# B&R Automation Studio project A2019059_Linka_Power_CP (part 38)

#### TesterKomunikacia.st
```iecst
ACTION TesterKomunikacia:

	//Vstupy z Testera do PLC//
	AteqLeakageTester_A.Stav_RESET_DONE:= AteqLeakageTester_A.Profinet_PLC_INPUTS[1].0;
	AteqLeakageTester_A.Stav_START_DONE:= AteqLeakageTester_A.Profinet_PLC_INPUTS[1].1;
	AteqLeakageTester_A.Stav_ZmenaProgramu_DONE:= AteqLeakageTester_A.Profinet_PLC_INPUTS[1].3;
	AteqLeakageTester_A.Stav_CitanieParametrov_OK:= AteqLeakageTester_A.Profinet_PLC_INPUTS[1].5;

    AteqLeakageTester_A.Stav_CitanieParametrov_ERROR:= AteqLeakageTester_A.Profinet_PLC_INPUTS[3].5;

	AteqLeakageTester_A.CisloAktualnehoProgramu.0:= AteqLeakageTester_A.Profinet_PLC_INPUTS[7].0;
	AteqLeakageTester_A.CisloAktualnehoProgramu.1:= AteqLeakageTester_A.Profinet_PLC_INPUTS[7].1;
	AteqLeakageTester_A.CisloAktualnehoProgramu.2:= AteqLeakageTester_A.Profinet_PLC_INPUTS[7].2;
	AteqLeakageTester_A.CisloAktualnehoProgramu.3:= AteqLeakageTester_A.Profinet_PLC_INPUTS[7].3;
	AteqLeakageTester_A.CisloAktualnehoProgramu.4:= AteqLeakageTester_A.Profinet_PLC_INPUTS[7].4;
	AteqLeakageTester_A.CisloAktualnehoProgramu.5:= AteqLeakageTester_A.Profinet_PLC_INPUTS[7].5;
	AteqLeakageTester_A.CisloAktualnehoProgramu.6:= AteqLeakageTester_A.Profinet_PLC_INPUTS[7].6;
	AteqLeakageTester_A.CisloAktualnehoProgramu.7:= AteqLeakageTester_A.Profinet_PLC_INPUTS[7].7;

	AteqLeakageTester_A.CisloAktualnehoProgramu.8:= AteqLeakageTester_A.Profinet_PLC_INPUTS[8].0;
	AteqLeakageTester_A.CisloAktualnehoProgramu.9:= AteqLeakageTester_A.Profinet_PLC_INPUTS[8].1;
	AteqLeakageTester_A.CisloAktualnehoProgramu.10:= AteqLeakageTester_A.Profinet_PLC_INPUTS[8].2;
	AteqLeakageTester_A.CisloAktualnehoProgramu.11:= AteqLeakageTester_A.Profinet_PLC_INPUTS[8].3;
	AteqLeakageTester_A.CisloAktualnehoProgramu.12:= AteqLeakageTester_A.Profinet_PLC_INPUTS[8].4;
	AteqLeakageTester_A.CisloAktualnehoProgramu.13:= AteqLeakageTester_A.Profinet_PLC_INPUTS[8].5;
	AteqLeakageTester_A.CisloAktualnehoProgramu.14:= AteqLeakageTester_A.Profinet_PLC_INPUTS[8].6;
	AteqLeakageTester_A.CisloAktualnehoProgramu.15:= AteqLeakageTester_A.Profinet_PLC_INPUTS[8].7;

	AteqLeakageTester_A.VysledokTestovania_OK:= AteqLeakageTester_A.Profinet_PLC_INPUTS[13].0;
	AteqLeakageTester_A.VysledokTestovania_NG:= AteqLeakageTester_A.Profinet_PLC_INPUTS[13].1;
	AteqLeakageTester_A.Stav_ERROR:= AteqLeakageTester_A.Profinet_PLC_INPUTS[13].3;
	AteqLeakageTester_A.Stav_READY:= AteqLeakageTester_A.Profinet_PLC_INPUTS[13].5;

    AteqLeakageTester_A.ReadParameter_1.0:= AteqLeakageTester_A.Profinet_PLC_INPUTS[35].0;
    AteqLeakageTester_A.ReadParameter_1.1:= AteqLeakageTester_A.Profinet_PLC_INPUTS[35].1;
    AteqLeakageTester_A.ReadParameter_1.2:= AteqLeakageTester_A.Profinet_PLC_INPUTS[35].2;
    AteqLeakageTester_A.ReadParameter_1.3:= AteqLeakageTester_A.Profinet_PLC_INPUTS[35].3;
    AteqLeakageTester_A.ReadParameter_1.4:= AteqLeakageTester_A.Profinet_PLC_INPUTS[35].4;
    AteqLeakageTester_A.ReadParameter_1.5:= AteqLeakageTester_A.Profinet_PLC_INPUTS[35].5;
    AteqLeakageTester_A.ReadParameter_1.6:= AteqLeakageTester_A.Profinet_PLC_INPUTS[35].6;
    AteqLeakageTester_A.ReadParameter_1.7:= AteqLeakageTester_A.Profinet_PLC_INPUTS[35].7;
    AteqLeakageTester_A.ReadParameter_1.8:= AteqLeakageTester_A.Profinet_PLC_INPUTS[36].0;
    AteqLeakageTester_A.ReadParameter_1.9:= AteqLeakageTester_A.Profinet_PLC_INPUTS[36].1;
    AteqLeakageTester_A.ReadParameter_1.10:= AteqLeakageTester_A.Profinet_PLC_INPUTS[36].2;
    AteqLeakageTester_A.ReadParameter_1.11:= AteqLeakageTester_A.Profinet_PLC_INPUTS[36].3;
    AteqLeakageTester_A.ReadParameter_1.12:= AteqLeakageTester_A.Profinet_PLC_INPUTS[36].4;
    AteqLeakageTester_A.ReadParameter_1.13:= AteqLeakageTester_A.Profinet_PLC_INPUTS[36].5;
    AteqLeakageTester_A.ReadParameter_1.14:= AteqLeakageTester_A.Profinet_PLC_INPUTS[36].6;
    AteqLeakageTester_A.ReadParameter_1.15:= AteqLeakageTester_A.Profinet_PLC_INPUTS[36].7;

    AteqLeakageTester_A.ReadParameter_2.0:= AteqLeakageTester_A.Profinet_PLC_INPUTS[41].0;
    AteqLeakageTester_A.ReadParameter_2.1:= AteqLeakageTester_A.Profinet_PLC_INPUTS[41].1;
    AteqLeakageTester_A.ReadParameter_2.2:= AteqLeakageTester_A.Profinet_PLC_INPUTS[41].2;
    AteqLeakageTester_A.ReadParameter_2.3:= AteqLeakageTester_A.Profinet_PLC_INPUTS[41].3;
    AteqLeakageTester_A.ReadParameter_2.4:= AteqLeakageTester_A.Profinet_PLC_INPUTS[41].4;
    AteqLeakageTester_A.ReadParameter_2.5:= AteqLeakageTester_A.Profinet_PLC_INPUTS[41].5;
    AteqLeakageTester_A.ReadParameter_2.6:= AteqLeakageTester_A.Profinet_PLC_INPUTS[41].6;
    AteqLeakageTester_A.ReadParameter_2.7:= AteqLeakageTester_A.Profinet_PLC_INPUTS[41].7;
    AteqLeakageTester_A.ReadParameter_2.8:= AteqLeakageTester_A.Profinet_PLC_INPUTS[42].0;
    AteqLeakageTester_A.ReadParameter_2.9:= AteqLeakageTester_A.Profinet_PLC_INPUTS[42].1;
    AteqLeakageTester_A.ReadParameter_2.10:= AteqLeakageTester_A.Profinet_PLC_INPUTS[42].2;
    AteqLeakageTester_A.ReadParameter_2.11:= AteqLeakageTester_A.Profinet_PLC_INPUTS[42].3;
    AteqLeakageTester_A.ReadParameter_2.12:= AteqLeakageTester_A.Profinet_PLC_INPUTS[42].4;
    AteqLeakageTester_A.ReadParameter_2.13:= AteqLeakageTester_A.Profinet_PLC_INPUTS[42].5;
    AteqLeakageTester_A.ReadParameter_2.14:= AteqLeakageTester_A.Profinet_PLC_INPUTS[42].6;
    AteqLeakageTester_A.ReadParameter_2.15:= AteqLeakageTester_A.Profinet_PLC_INPUTS[42].7;

    AteqLeakageTester_A.ReadParameter_3.0:= AteqLeakageTester_A.Profinet_PLC_INPUTS[47].0;
    AteqLeakageTester_A.ReadParameter_3.1:= AteqLeakageTester_A.Profinet_PLC_INPUTS[47].1;
    AteqLeakageTester_A.ReadParameter_3.2:= AteqLeakageTester_A.Profinet_PLC_INPUTS[47].2;
    AteqLeakageTester_A.ReadParameter_3.3:= AteqLeakageTester_A.Profinet_PLC_INPUTS[47].3;
    AteqLeakageTester_A.ReadParameter_3.4:= AteqLeakageTester_A.Profinet_PLC_INPUTS[47].4;
    AteqLeakageTester_A.ReadParameter_3.5:= AteqLeakageTester_A.Profinet_PLC_INPUTS[47].5;
    AteqLeakageTester_A.ReadParameter_3.6:= AteqLeakageTester_A.Profinet_PLC_INPUTS[47].6;
    AteqLeakageTester_A.ReadParameter_3.7:= AteqLeakageTester_A.Profinet_PLC_INPUTS[47].7;
    AteqLeakageTester_A.ReadParameter_3.8:= AteqLeakageTester_A.Profinet_PLC_INPUTS[48].0;
    AteqLeakageTester_A.ReadParameter_3.9:= AteqLeakageTester_A.Profinet_PLC_INPUTS[48].1;
    AteqLeakageTester_A.ReadParameter_3.10:= AteqLeakageTester_A.Profinet_PLC_INPUTS[48].2;
    AteqLeakageTester_A.ReadParameter_3.11:= AteqLeakageTester_A.Profinet_PLC_INPUTS[48].3;
    AteqLeakageTester_A.ReadParameter_3.12:= AteqLeakageTester_A.Profinet_PLC_INPUTS[48].4;
    AteqLeakageTester_A.ReadParameter_3.13:= AteqLeakageTester_A.Profinet_PLC_INPUTS[48].5;
    AteqLeakageTester_A.ReadParameter_3.14:= AteqLeakageTester_A.Profinet_PLC_INPUTS[48].6;
    AteqLeakageTester_A.ReadParameter_3.15:= AteqLeakageTester_A.Profinet_PLC_INPUTS[48].7;

    AteqLeakageTester_A.ReadParameter_4.0:= AteqLeakageTester_A.Profinet_PLC_INPUTS[53].0;
    AteqLeakageTester_A.ReadParameter_4.1:= AteqLeakageTester_A.Profinet_PLC_INPUTS[53].1;
    AteqLeakageTester_A.ReadParameter_4.2:= AteqLeakageTester_A.Profinet_PLC_INPUTS[53].2;
    AteqLeakageTester_A.ReadParameter_4.3:= AteqLeakageTester_A.Profinet_PLC_INPUTS[53].3;
    AteqLeakageTester_A.ReadParameter_4.4:= AteqLeakageTester_A.Profinet_PLC_INPUTS[53].4;
    AteqLeakageTester_A.ReadParameter_4.5:= AteqLeakageTester_A.Profinet_PLC_INPUTS[53].5;
    AteqLeakageTester_A.ReadParameter_4.6:= AteqLeakageTester_A.Profinet_PLC_INPUTS[53].6;
    AteqLeakageTester_A.ReadParameter_4.7:= AteqLeakageTester_A.Profinet_PLC_INPUTS[53].7;
    AteqLeakageTester_A.ReadParameter_4.8:= AteqLeakageTester_A.Profinet_PLC_INPUTS[54].0;
    AteqLeakageTester_A.ReadParameter_4.9:= AteqLeakageTester_A.Profinet_PLC_INPUTS[54].1;
    AteqLeakageTester_A.ReadParameter_4.10:= AteqLeakageTester_A.Profinet_PLC_INPUTS[54].2;
    AteqLeakageTester_A.ReadParameter_4.11:= AteqLeakageTester_A.Profinet_PLC_INPUTS[54].3;
    AteqLeakageTester_A.ReadParameter_4.12:= AteqLeakageTester_A.Profinet_PLC_INPUTS[54].4;
    AteqLeakageTester_A.ReadParameter_4.13:= AteqLeakageTester_A.Profinet_PLC_INPUTS[54].5;
    AteqLeakageTester_A.ReadParameter_4.14:= AteqLeakageTester_A.Profinet_PLC_INPUTS[54].6;
    AteqLeakageTester_A.ReadParameter_4.15:= AteqLeakageTester_A.Profinet_PLC_INPUTS[54].7;

    AteqLeakageTester_A.ReadParameter_5.0:= AteqLeakageTester_A.Profinet_PLC_INPUTS[24].0;
    AteqLeakageTester_A.ReadParameter_5.1:= AteqLeakageTester_A.Profinet_PLC_INPUTS[24].1;
    AteqLeakageTester_A.ReadParameter_5.2:= AteqLeakageTester_A.Profinet_PLC_INPUTS[24].2;
    AteqLeakageTester_A.ReadParameter_5.3:= AteqLeakageTester_A.Profinet_PLC_INPUTS[24].3;
    AteqLeakageTester_A.ReadParameter_5.4:= AteqLeakageTester_A.Profinet_PLC_INPUTS[24].4;
    AteqLeakageTester_A.ReadParameter_5.5:= AteqLeakageTester_A.Profinet_PLC_INPUTS[24].5;
    AteqLeakageTester_A.ReadParameter_5.6:= AteqLeakageTester_A.Profinet_PLC_INPUTS[24].6;
    AteqLeakageTester_A.ReadParameter_5.7:= AteqLeakageTester_A.Profinet_PLC_INPUTS[24].7;
    AteqLeakageTester_A.ReadParameter_5.8:= AteqLeakageTester_A.Profinet_PLC_INPUTS[25].0;
    AteqLeakageTester_A.ReadParameter_5.9:= AteqLeakageTester_A.Profinet_PLC_INPUTS[25].1;
    AteqLeakageTester_A.ReadParameter_5.10:= AteqLeakageTester_A.Profinet_PLC_INPUTS[25].2;
    AteqLeakageTester_A.ReadParameter_5.11:= AteqLeakageTester_A.Profinet_PLC_INPUTS[25].3;
    AteqLeakageTester_A.ReadParameter_5.12:= AteqLeakageTester_A.Profinet_PLC_INPUTS[25].4;
    AteqLeakageTester_A.ReadParameter_5.13:= AteqLeakageTester_A.Profinet_PLC_INPUTS[25].5;
    AteqLeakageTester_A.ReadParameter_5.14:= AteqLeakageTester_A.Profinet_PLC_INPUTS[25].6;
    AteqLeakageTester_A.ReadParameter_5.15:= AteqLeakageTester_A.Profinet_PLC_INPUTS[25].7;
    AteqLeakageTester_A.ReadParameter_5.16:= AteqLeakageTester_A.Profinet_PLC_INPUTS[26].0;
    AteqLeakageTester_A.ReadParameter_5.17:= AteqLeakageTester_A.Profinet_PLC_INPUTS[26].1;
    AteqLeakageTester_A.ReadParameter_5.18:= AteqLeakageTester_A.Profinet_PLC_INPUTS[26].2;
    AteqLeakageTester_A.ReadParameter_5.19:= AteqLeakageTester_A.Profinet_PLC_INPUTS[26].3;
    AteqLeakageTester_A.ReadParameter_5.20:= AteqLeakageTester_A.Profinet_PLC_INPUTS[26].4;
    AteqLeakageTester_A.ReadParameter_5.21:= AteqLeakageTester_A.Profinet_PLC_INPUTS[26].5;
    AteqLeakageTester_A.ReadParameter_5.22:= AteqLeakageTester_A.Profinet_PLC_INPUTS[26].6;
    AteqLeakageTester_A.ReadParameter_5.23:= AteqLeakageTester_A.Profinet_PLC_INPUTS[26].7;
    AteqLeakageTester_A.ReadParameter_5.24:= AteqLeakageTester_A.Profinet_PLC_INPUTS[27].0;
    AteqLeakageTester_A.ReadParameter_5.25:= AteqLeakageTester_A.Profinet_PLC_INPUTS[27].1;
    AteqLeakageTester_A.ReadParameter_5.26:= AteqLeakageTester_A.Profinet_PLC_INPUTS[27].2;
    AteqLeakageTester_A.ReadParameter_5.27:= AteqLeakageTester_A.Profinet_PLC_INPUTS[27].3;
    AteqLeakageTester_A.ReadParameter_5.28:= AteqLeakageTester_A.Profinet_PLC_INPUTS[27].4;
    AteqLeakageTester_A.ReadParameter_5.29:= AteqLeakageTester_A.Profinet_PLC_INPUTS[27].5;
    AteqLeakageTester_A.ReadParameter_5.30:= AteqLeakageTester_A.Profinet_PLC_INPUTS[27].6;
    AteqLeakageTester_A.ReadParameter_5.31:= AteqLeakageTester_A.Profinet_PLC_INPUTS[27].7;

	//Vystupy z PLC do Testera//
	AteqLeakageTester_A.Profinet_PLC_OUTPUTS[1].0:= AteqLeakageTester_A.RESET_Vysledkov;
	AteqLeakageTester_A.Profinet_PLC_OUTPUTS[1].1:= AteqLeakageTester_A.START_Testovania;
	AteqLeakageTester_A.Profinet_PLC_OUTPUTS[1].3:= AteqLeakageTester_A.ZMEN_Program;
	AteqLeakageTester_A.Profinet_PLC_OUTPUTS[1].5:= AteqLeakageTester_A.CitajParametreTestera;

	AteqLeakageTester_A.Profinet_PLC_OUTPUTS[7].0:= AteqLeakageTester_A.CisloZadanehoProgramu.0;
	AteqLeakageTester_A.Profinet_PLC_OUTPUTS[7].1:= AteqLeakageTester_A.CisloZadanehoProgramu.1;
	AteqLeakageTester_A.Profinet_PLC_OUTPUTS[7].2:= AteqLeakageTester_A.CisloZadanehoProgramu.2;
	AteqLeakageTester_A.Profinet_PLC_OUTPUTS[7].3:= AteqLeakageTester_A.CisloZadanehoProgramu.3;
	AteqLeakageTester_A.Profinet_PLC_OUTPUTS[7].4:= AteqLeakageTester_A.CisloZadanehoProgramu.4;
	AteqLeakageTester_A.Profinet_PLC_OUTPUTS[7].5:= AteqLeakageTester_A.CisloZadanehoProgramu.5;
	AteqLeakageTester_A.Profinet_PLC_OUTPUTS[7].6:= AteqLeakageTester_A.CisloZadanehoProgramu.6;
	AteqLeakageTester_A.Profinet_PLC_OUTPUTS[7].7:= AteqLeakageTester_A.CisloZadanehoProgramu.7;

	AteqLeakageTester_A.Profinet_PLC_OUTPUTS[8].0:= AteqLeakageTester_A.CisloZadanehoProgramu.8;
	AteqLeakageTester_A.Profinet_PLC_OUTPUTS[8].1:= AteqLeakageTester_A.CisloZadanehoProgramu.9;
	AteqLeakageTester_A.Profinet_PLC_OUTPUTS[8].2:= AteqLeakageTester_A.CisloZadanehoProgramu.10;
	AteqLeakageTester_A.Profinet_PLC_OUTPUTS[8].3:= AteqLeakageTester_A.CisloZadanehoProgramu.11;
	AteqLeakageTester_A.Profinet_PLC_OUTPUTS[8].4:= AteqLeakageTester_A.CisloZadanehoProgramu.12;
	AteqLeakageTester_A.Profinet_PLC_OUTPUTS[8].5:= AteqLeakageTester_A.CisloZadanehoProgramu.13;
	AteqLeakageTester_A.Profinet_PLC_OUTPUTS[8].6:= AteqLeakageTester_A.CisloZadanehoProgramu.14;
	AteqLeakageTester_A.Profinet_PLC_OUTPUTS[8].7:= AteqLeakageTester_A.CisloZadanehoProgramu.15;

	AteqLeakageTester_A.PocetCitanychParametrov:= 4;
    AteqLeakageTester_A.IdentifikaciaParametra_1:= 1;
    AteqLeakageTester_A.IdentifikaciaParametra_2:= 2;
    AteqLeakageTester_A.IdentifikaciaParametra_3:= 66;
    AteqLeakageTester_A.IdentifikaciaParametra_4:= 60;

    //Vyčítané parametre//
    CasPneniaREAL:= UINT_TO_REAL(AteqLeakageTester_A.ReadParameter_1);
    AteqLeakageTester_A.CasPnenia:= CasPneniaREAL/1000;
    CasStabilizacieREAL:= UINT_TO_REAL(AteqLeakageTester_A.ReadParameter_2);
    AteqLeakageTester_A.CasStabilizacie:= CasStabilizacieREAL/1000;
    TlakPlneniaREAL:= UINT_TO_REAL(AteqLeakageTester_A.ReadParameter_3);
    AteqLeakageTester_A.TlakPlnenia:= TlakPlneniaREAL/1000;
    ToleranciaREAL:= UINT_TO_REAL(AteqLeakageTester_A.ReadParameter_4);
    AteqLeakageTester_A.Tolerancia:= ToleranciaREAL/1000;
    TlakUnikuREAL:= DINT_TO_REAL(AteqLeakageTester_A.ReadParameter_5);
    AteqLeakageTester_A.TlakUniku:= ((TlakUnikuREAL/1000)*6)/1536;

END_ACTION
```

### Program Logical/Program/Pracovisko_3/P3_StoperLeakageTestB (IEC)

#### Main.st - Init, cyclic, exit code
```iecst
PROGRAM _INIT
    Triger_0:= FALSE;
    Triger_1:= FALSE;

    P3_LeakageTestB.STAV.Tester_ON:= TRUE;
END_PROGRAM

PROGRAM _CYCLIC

	//Volanie podprogramov//
    OvlCentrovacky;
    IOLinkKomunikacia;
    OvlPritlaku;
    TesterKomunikacia;

    //Volanie funkcie SequenceControl//
    SequenceControl(SC:= SC_P3_LeakageTestB);

    //Príznak leakage test B východzia pozícia//
    IF P3_LeakageTestB.IN.Centrovanie_ZASUNUTE_IS74 AND P3_LeakageTestB.IN.Pritlak_ZASUNUTY_MS48 AND P3_LeakageTestB.IN.Kopito_ZASUNUTE_IS70 THEN
        P3_LeakageTestB_VychodziaPozicia:= TRUE;
    ELSE
        P3_LeakageTestB_VychodziaPozicia:= FALSE;
    END_IF

    //Reset sekcie //
    IF P3_LeakageTestB.Reset THEN
        SC_P3_LeakageTestB.Step:= 0;
        P3_LeakageTestB.Reset:= FALSE;
    END_IF

    IF NOT Safety.STAV.P3_ZonaBunky_AKTIVNA AND NOT P3_LeakageTestB.Automat THEN
        SC_P3_LeakageTestB.Step:= 0;
    END_IF

    IF NOT Safety.STAV.P3_ZonaBunky_AKTIVNA AND NOT Triger_0 THEN
        Triger_0:= TRUE;
        IF P3_LeakageTestB.IN.PritomnostPaletky_S24 AND P3_LeakageTestB.Automat THEN
            IF NOT Paletka[i].VnutornyStav.KomunikaciaOtvorena THEN
                SC_P3_LeakageTestB.ResetStep:= TRUE;
                SC_P3_LeakageTestB.Step:= 0;
            ELSIF Paletka[i].VnutornyStav.KomunikaciaUzavreta THEN
                SC_P3_LeakageTestB.ResetStep:= TRUE;
                SC_P3_LeakageTestB.Step:= 0;
            ELSIF Paletka[i].VnutornyStav.KomunikaciaOtvorena THEN
                Paletka[i].PAR.StavPowerCP:= 'FAIL';
                Paletka[i].PAR.StavPaletky:= 'NG';
                P3_LeakageTestB.KoniecCyklu:= TRUE;
                SC_P3_LeakageTestB.ResetStep:= TRUE;
                SC_P3_LeakageTestB.Step:= 550;
            END_IF
        END_IF
    END_IF

    IF Safety.STAV.P3_ZonaBunky_AKTIVNA THEN
        Triger_0:= FALSE;
    END_IF

    //Porucha stanice//
    IF P3_PoruchaST3 AND NOT Triger_1  THEN
        Triger_1:= TRUE;
        IF P3_LeakageTestB.IN.PritomnostPaletky_S24 AND P3_LeakageTestB.Automat THEN
            IF NOT Paletka[i].VnutornyStav.KomunikaciaOtvorena THEN
                SC_P3_LeakageTestB.ResetStep:= TRUE;
                SC_P3_LeakageTestB.Step:= 0;
            ELSIF Paletka[i].VnutornyStav.KomunikaciaUzavreta THEN
                SC_P3_LeakageTestB.ResetStep:= TRUE;
                SC_P3_LeakageTestB.Step:= 0;
            ELSIF Paletka[i].VnutornyStav.KomunikaciaOtvorena THEN
                Paletka[i].PAR.StavPowerCP:= 'FAIL';
                Paletka[i].PAR.StavPaletky:= 'NG';
                P3_LeakageTestB.KoniecCyklu:= TRUE;
                SC_P3_LeakageTestB.ResetStep:= TRUE;
                SC_P3_LeakageTestB.Step:= 550;
            END_IF
        ELSE
            SC_P3_LeakageTestB.ResetStep:= TRUE;
            SC_P3_LeakageTestB.Step:= 0;
        END_IF
    END_IF

    IF NOT P3_PoruchaST3 THEN
        Triger_1:= FALSE;
    END_IF

    CASE SC_P3_LeakageTestB.Step OF

        0:
            SC_P3_LeakageTestB.StepName:='0 - Nulovanie';
            SC_OvlCentrovacky.Step:= 0;
            SC_OvlPritlaku.Step:= 0;
            P3_LeakageTestB.Automat:= FALSE;
            P3_LeakageTestB.KoniecCyklu:= FALSE;
            P3_LeakageTestB.Manual:= FALSE;
            P3_LeakageTestB.STAV.PoINIT:= FALSE;
            P3_LeakageTestB.OUT.Kopito_VYSUN_YV145:= FALSE;
            P3_LeakageTestB.OUT.Kopito_ZASUN_YV146:= TRUE;
            P3_LeakageTestB.OUT.ZasunStoper_YV135:= FALSE;
            (*P3_LeakageTestB.OUT.PneuZamok_ODOMKNI_YV160:= FALSE;*)
            P3_LeakageTestB.STAV.KOM_PLC_OdoslanieFotiek_OK:= FALSE;
            P3_LeakageTestB.STAV.KOM_PLC_VymazanieFotiek_OK:= FALSE;
            TRCB_P3_LeakageTestB_ST8B.CMD.VyziadajStavPaletky_TYP1:= FALSE;
            TRCB_P3_LeakageTestB_ST8B.CMD.PriradQRkodFiltra_TYP3:= FALSE;
            TRCB_P3_LeakageTestB_ST8B.CMD.OdosliStavPaletky_TYP2:= FALSE;
            AteqLeakageTester_B.CitajParametreTestera:= FALSE;
            PrecitaneCisloPaletky:= '';
            AteqLeakageTester_B.START_Testovania:= FALSE;
            PocetDopytovNaServer:= 0;
            Taktime_LeakageTestB_ST8B.CMD.START_Merania_1:= FALSE;
            Taktime_LeakageTestB_ST8B.CMD.START_Merania_2:= FALSE;
            P3_LeakageTestB.STAV.PrebiehaVyvezeniePaletky:= FALSE;
            TestovaciKus:= FALSE;
            Revork:= FALSE;
            P3_LeakageTestB.OUT.KOM_StanicaA_StartTestovania:= FALSE;
            P3_LeakageTestB.RR_TestovanieLeakageTestu:= FALSE;
            P3_LeakageTestB.RR_VysunSpodneKopito:= FALSE;
            P3_LeakageTestB.RR_TestovaciaSekvencia:= FALSE;
            P3_LeakageTestB.STAV.TestovaciaSekvencia_BUSY:= FALSE;
            PocetOpakovaniTestu:= 0;
            OpakovanyTest:= FALSE;
            P34_Vizu.ZobrazHL2_ST8:= FALSE;
            TRCB_P3_LeakTestB_OpatovnyDopyt:= FALSE;
            TRCB_P3_LeakTestB_PaletkaNG:= FALSE;

            IF Safety.STAV.P3_ZonaBunky_AKTIVNA AND NOT P3_Pracovisko.STAV.PORUCHA AND P3_Pracovisko.IN.PrivodVzduchu_SnimacTlaku_S25 THEN
                SC_P3_LeakageTestB.ResetStep:= TRUE;
                SC_P3_LeakageTestB.Step:= 1;
            END_IF

        1:
            SC_P3_LeakageTestB.StepName:='1 - Cakam na spustenie vyroby';
            P3_LeakageTestB.KoniecCyklu:= FALSE;
            IF P3_LeakageTestB.Automat THEN
                SC_P3_LeakageTestB.Step:= 2;
            ELSIF P3_LeakageTestB.Manual THEN
                SC_P3_LeakageTestB.Step:= 700;
            END_IF

            //********************************************************Inicializácia****************************************************************************//

        2:
            SC_P3_LeakageTestB.StepName:='2 - Inicializacia - cakam na spustenie inicializacie';
            SC_P3_LeakageTestB.IdleTime.PT:= T#2s;
            SC_P3_LeakageTestB.AlarmTime.PT:= T#5s;

            SC_P3_LeakageTestB.IdleTime.IN:= TRUE;

            IF SC_P3_LeakageTestB.IdleTime.Q THEN
                SC_P3_LeakageTestB.ResetStep:= TRUE;
                SC_P3_LeakageTestB.Step:= 3;
            END_IF

        3:
            SC_P3_LeakageTestB.StepName:='3 - Inicializacia - zasunutie pritlaku';
            SC_P3_LeakageTestB.IdleTime.PT:= T#2s;
            SC_P3_LeakageTestB.AlarmTime.PT:= T#5s;

            IF NOT SC_P3_LeakageTestB.Switch1 THEN
                P3_LeakageTestB.OUT.PneuZamok_ODOMKNI_YV160:= TRUE;
                Pritlak_ZASUN:= TRUE;
                SC_P3_LeakageTestB.Switch1:= TRUE;
            END_IF

            IF P3_LeakageTestB.IN.Pritlak_ZASUNUTY_MS48 THEN
                P3_LeakageTestB.OUT.PneuZamok_ODOMKNI_YV160:= FALSE;
                SC_P3_LeakageTestB.ResetStep:= TRUE;
                SC_P3_LeakageTestB.Step:= 8;
            END_IF

        8:
            SC_P3_LeakageTestB.StepName:='8 - Inicializacia - zasunutie centrovacky';
            SC_P3_LeakageTestB.IdleTime.PT:= T#4s;
            SC_P3_LeakageTestB.AlarmTime.PT:= T#5s;

            IF NOT SC_P3_LeakageTestB.Switch1 THEN
                Centrovacku_ZASUN:= TRUE;
                SC_P3_LeakageTestB.Switch1:= TRUE;
            END_IF

            IF P3_LeakageTestB.IN.Centrovanie_ZASUNUTE_IS74 AND P3_Dopravniky.STAV.PoINIT THEN
                SC_P3_LeakageTestB.ResetStep:= TRUE;
                SC_P3_LeakageTestB.Step:= 10;
            END_IF

        10:
            SC_P3_LeakageTestB.StepName:='10 - Inicializacia - kontrola typu zalozeneho kopita';
            SC_P3_LeakageTestB.IdleTime.PT:= T#4s;
            SC_P3_LeakageTestB.AlarmTime.PT:= T#5s;

            IF Linka.PAR.ZvolenyModel = '4F' AND P3_LeakageTestB.IN.PritomnostKopita_IS69 AND P3_LeakageTestB.IN.Tester_TypKonektoru_4F THEN
                SC_P3_LeakageTestB.ResetStep:= TRUE;
                SC_P3_LeakageTestB.Step:= 13;
            ELSIF Linka.PAR.ZvolenyModel = '5F' AND P3_LeakageTestB.IN.PritomnostKopita_IS69 AND P3_LeakageTestB.IN.Tester_TypKonektoru_5F_5H THEN
                SC_P3_LeakageTestB.ResetStep:= TRUE;
                SC_P3_LeakageTestB.Step:= 13;
            ELSIF Linka.PAR.ZvolenyModel = '5H' AND P3_LeakageTestB.IN.PritomnostKopita_IS69 AND P3_LeakageTestB.IN.Tester_TypKonektoru_5F_5H THEN
                SC_P3_LeakageTestB.ResetStep:= TRUE;
                SC_P3_LeakageTestB.Step:= 13;
            ELSE
                P34_Alarmy[315]:= TRUE;
                P3_PoruchaST3:= TRUE;
            END_IF

        13:
            SC_P3_LeakageTestB.StepName:='13 - Inicializacia - hladanie paletky';
            SC_P3_LeakageTestB.IdleTime.PT:= T#5s;
            SC_P3_LeakageTestB.AlarmTime.PT:= T#5s;
            SC_P3_LeakageTestB.IdleTime.IN:= TRUE;

            IF P3_LeakageTestB.IN.PritomnostPaletky_S24 THEN
                P3_LeakageTestA.STAV.PrebiehaVyvezeniePaletky:= FALSE;
                SC_P3_LeakageTestB.ResetStep:= TRUE;
                SC_P3_LeakageTestB.Step:= 20;
            ELSIF SC_P3_LeakageTestB.IdleTime.Q THEN
                P3_LeakageTestB.STAV.PoINIT:= TRUE;
                SC_P3_LeakageTestB.ResetStep:= TRUE;
                SC_P3_LeakageTestB.Step:= 100;
            END_IF

        20:
            SC_P3_LeakageTestB.StepName:='20 - Inicializacia - precitanie cisla paletky';
            SC_P3_LeakageTestB.IdleTime.PT:= T#200ms;
            SC_P3_LeakageTestB.AlarmTime.PT:= T#5s;
            SC_P3_LeakageTestB.IdleTime.IN:= TRUE;

            IF SC_P3_LeakageTestB.IdleTime.Q THEN
                PrecitaneCisloPaletky:= USINT_TO_STRING(P3_LeakageTestB.IN.PrecitaneCisloPaletky_S24);
                i:= 0;
                SC_P3_LeakageTestB.ResetStep:= TRUE;
                SC_P3_LeakageTestB.Step:= 23;
            END_IF

        23:
            SC_P3_LeakageTestB.StepName:='23 - Inicializacia - priradenie indexu paletky na zaklade precitanej hodnoty';
            SC_P3_LeakageTestB.IdleTime.PT:= T#200ms;
            SC_P3_LeakageTestB.AlarmTime.PT:= T#5s;

            IF PrecitaneCisloPaletky = '171' THEN
                i:= 1;
            ELSIF PrecitaneCisloPaletky = '164' THEN
                i:= 2;
            ELSIF PrecitaneCisloPaletky = '181' THEN
                i:= 3;
            ELSIF PrecitaneCisloPaletky = '168' THEN
                i:= 4;
            ELSIF PrecitaneCisloPaletky = '140' THEN
                i:= 5;
            ELSIF PrecitaneCisloPaletky = '110' THEN
                i:= 6;
            ELSIF PrecitaneCisloPaletky = '156' THEN
                i:= 7;
            ELSIF PrecitaneCisloPaletky = '127' THEN
                i:= 8;
            ELSIF PrecitaneCisloPaletky = '139' THEN
                i:= 9;
            ELSIF PrecitaneCisloPaletky = '131' THEN
                i:= 10;
            ELSIF PrecitaneCisloPaletky = '178' THEN
                i:= 11;
            ELSIF PrecitaneCisloPaletky = '206' THEN
                i:= 12;
            ELSIF PrecitaneCisloPaletky = '119' THEN
                i:= 13;
            ELSIF PrecitaneCisloPaletky = '163' THEN
                i:= 14;
            ELSIF PrecitaneCisloPaletky = '128' THEN
                i:= 15;
            ELSIF PrecitaneCisloPaletky = '175' THEN
                i:= 16;
            ELSIF PrecitaneCisloPaletky = '138' THEN
                i:= 17;
            ELSE
                P34_Alarmy[312]:= TRUE;
                P3_PoruchaST3:= TRUE;
            END_IF

            IF i<> 0 THEN
                Paletka[i].PAR.CisloPaletky:= USINT_TO_STRING(i);
                P3_LeakageTestB.PAR.IndexPaletky_STRING:= USINT_TO_STRING(i);
                P3_LeakageTestB.PAR.IndexPaletky:= i;
                PrecitaneCisloPaletky:= '';
                SC_P3_LeakageTestB.ResetStep:= TRUE;
                SC_P3_LeakageTestB.Step:= 30;
            END_IF

        30:
            SC_P3_LeakageTestB.StepName:='30 - Inicializacia - kontrola stavu paletky';
            SC_P3_LeakageTestB.IdleTime.PT:= T#200ms;
            SC_P3_LeakageTestB.AlarmTime.PT:= T#5s;

            IF Paletka[i].PAR.TestovaciKus AND Paletka[i].PAR.CisloTestovacejStanice = 'ST_8A,8B' THEN
                IF P3_LeakageTestB.STAV.Tester_ON THEN
                    TestovaciKus:= TRUE;
                    P3_LeakageTestB.STAV.PoINIT:= TRUE;
                    SC_P3_LeakageTestB.ResetStep:= TRUE;
                    SC_P3_LeakageTestB.Step:= 113;
                ELSE
                    P3_LeakageTestB.STAV.PoINIT:= TRUE;
                    SC_P3_LeakageTestB.ResetStep:= TRUE;
                    SC_P3_LeakageTestB.Step:= 560;
                END_IF
            ELSIF Paletka[i].PAR.TestovaciKus AND Paletka[i].PAR.CisloTestovacejStanice <> 'ST_8A,8B' THEN
                P3_LeakageTestB.STAV.PoINIT:= TRUE;
                SC_P3_LeakageTestB.ResetStep:= TRUE;
                SC_P3_LeakageTestB.Step:= 560;
            ELSIF Paletka[i].PAR.RevorkovyKus AND Paletka[i].PAR.CisloRevorkovejStanice = 'ST_8A,8B' THEN
                IF P3_LeakageTestB.STAV.Tester_ON THEN
                    Revork:= TRUE;
                    P3_LeakageTestB.STAV.PoINIT:= TRUE;
                    SC_P3_LeakageTestB.ResetStep:= TRUE;
                    SC_P3_LeakageTestB.Step:= 105;
                ELSE
                    P3_LeakageTestB.STAV.PoINIT:= TRUE;
                    SC_P3_LeakageTestB.ResetStep:= TRUE;
                    SC_P3_LeakageTestB.Step:= 560;
                END_IF
            ELSIF Paletka[i].PAR.RevorkovyKus AND Paletka[i].PAR.CisloRevorkovejStanice <> 'ST_8A,8B' THEN
                Revork:= FALSE;
                P3_LeakageTestB.STAV.PoINIT:= TRUE;
                SC_P3_LeakageTestB.ResetStep:= TRUE;
                SC_P3_LeakageTestB.Step:= 560;
            ELSIF Paletka[i].PAR.StavPaletky = 'OK' THEN
                SC_P3_LeakageTestB.ResetStep:= TRUE;
                SC_P3_LeakageTestB.Step:= 33;
            ELSIF Paletka[i].PAR.StavPaletky = 'NG' THEN
                P3_LeakageTestB.STAV.PoINIT:= TRUE;
                SC_P3_LeakageTestB.ResetStep:= TRUE;
                SC_P3_LeakageTestB.Step:= 560;
            END_IF

        33:
            SC_P3_LeakageTestB.StepName:='33 - Inicializacia - kontrola uzavretia komunikacie';
            SC_P3_LeakageTestB.IdleTime.PT:= T#200ms;
            SC_P3_LeakageTestB.AlarmTime.PT:= T#5s;

            IF Paletka[i].VnutornyStav.KomunikaciaUzavreta THEN
                P3_LeakageTestB.STAV.PoINIT:= TRUE;
                SC_P3_LeakageTestB.ResetStep:= TRUE;
                SC_P3_LeakageTestB.Step:= 560;
            ELSE
                SC_P3_LeakageTestB.ResetStep:= TRUE;
                SC_P3_LeakageTestB.Step:= 35;
            END_IF

        35:
            SC_P3_LeakageTestB.StepName:='35 - Inicializacia - kontrola otvorenia komunikacie';
            SC_P3_LeakageTestB.IdleTime.PT:= T#200ms;
            SC_P3_LeakageTestB.AlarmTime.PT:= T#5s;

            IF Paletka[i].VnutornyStav.KomunikaciaOtvorena THEN
                P3_LeakageTestB.STAV.PoINIT:= TRUE;
                SC_P3_LeakageTestB.ResetStep:= TRUE;
                SC_P3_LeakageTestB.Step:= 118;
            ELSE
                P3_LeakageTestB.STAV.PoINIT:= TRUE;
                SC_P3_LeakageTestB.ResetStep:= TRUE;
                SC_P3_LeakageTestB.Step:= 100;
            END_IF

            //********************************************************Automatický režim****************************************************************************//

        100:
            SC_P3_LeakageTestB.StepName:='100 - Automaticky Rezim - cakam na príchod paletky na stoper';
            SC_P3_LeakageTestB.IdleTime.PT:= T#200ms;
            SC_P3_LeakageTestB.AlarmTime.PT:= T#5s;

            IF P3_LeakageTestB.IN.PritomnostPaletky_S24 THEN
                P3_LeakageTestA.STAV.PrebiehaVyvezeniePaletky:= FALSE;
            END_IF

            SC_P3_LeakageTestB.IdleTime.IN:= P3_LeakageTestB.IN.PritomnostPaletky_S24;

            IF EDGEPOS(P3_LeakageTestB.IN.PritomnostPaletky_S24)THEN
                IF NOT Taktime_LeakageTestB_ST8B.CMD.START_Merania_1 THEN
                    Taktime_LeakageTestB_ST8B.CMD.START_Merania_1:= TRUE;
                ELSE
                    Taktime_LeakageTestB_ST8B.CMD.ZAPIS_Hodnot_1:= TRUE;
                END_IF
            END_IF

            IF P3_LeakageTestB.KoniecCyklu THEN
                SC_P3_LeakageTestB.ResetStep:= TRUE;
                SC_P3_LeakageTestB.Step:= 0;
            ELSIF SC_P3_LeakageTestB.IdleTime.Q THEN
                SC_P3_LeakageTestB.ResetStep:= TRUE;
                SC_P3_LeakageTestB.Step:= 101;
            END_IF

        101:
            SC_P3_LeakageTestB.StepName:='101 - Automaticky Rezim - precitanie cisla paletky';
            SC_P3_LeakageTestB.IdleTime.PT:= T#500ms;
            SC_P3_LeakageTestB.AlarmTime.PT:= T#5s;
            SC_P3_LeakageTestB.IdleTime.IN:= TRUE;

            PrecitaneCisloPaletky:= USINT_TO_STRING(P3_LeakageTestB.IN.PrecitaneCisloPaletky_S24);
            i:= 0;
            SC_P3_LeakageTestB.ResetStep:= TRUE;
            SC_P3_LeakageTestB.Step:= 102;

        102:
            SC_P3_LeakageTestB.StepName:='102 - Automaticky Rezim - priradenie indexu paletky na zaklade precitanej hodnoty';
            SC_P3_LeakageTestB.IdleTime.PT:= T#1s;
            SC_P3_LeakageTestB.AlarmTime.PT:= T#5s;

            IF PrecitaneCisloPaletky = '171' THEN
                i:= 1;
            ELSIF PrecitaneCisloPaletky = '164' THEN
                i:= 2;
            ELSIF PrecitaneCisloPaletky = '181' THEN
                i:= 3;
            ELSIF PrecitaneCisloPaletky = '168' THEN
                i:= 4;
            ELSIF PrecitaneCisloPaletky = '140' THEN
                i:= 5;
            ELSIF PrecitaneCisloPaletky = '110' THEN
                i:= 6;
            ELSIF PrecitaneCisloPaletky = '156' THEN
                i:= 7;
            ELSIF PrecitaneCisloPaletky = '127' THEN
                i:= 8;
            ELSIF PrecitaneCisloPaletky = '139' THEN
                i:= 9;
            ELSIF PrecitaneCisloPaletky = '131' THEN
                i:= 10;
            ELSIF PrecitaneCisloPaletky = '178' THEN
                i:= 11;
            ELSIF PrecitaneCisloPaletky = '206' THEN
                i:= 12;
            ELSIF PrecitaneCisloPaletky = '119' THEN
                i:= 13;
            ELSIF PrecitaneCisloPaletky = '163' THEN
                i:= 14;
            ELSIF PrecitaneCisloPaletky = '128' THEN
                i:= 15;
            ELSIF PrecitaneCisloPaletky = '175' THEN
                i:= 16;
            ELSIF PrecitaneCisloPaletky = '138' THEN
                i:= 17;
            ELSE
                P34_Alarmy[312]:= TRUE;
                P3_PoruchaST3:= TRUE;
            END_IF

            IF i<> 0 THEN
                Paletka[i].PAR.CisloPaletky:= USINT_TO_STRING(i);
                P3_LeakageTestB.PAR.IndexPaletky_STRING:= USINT_TO_STRING(i);
                P3_LeakageTestB.PAR.IndexPaletky:= i;
                PrecitaneCisloPaletky:= '';
                SC_P3_LeakageTestB.ResetStep:= TRUE;
                SC_P3_LeakageTestB.Step:= 103;
            END_IF

        103:
            SC_P3_LeakageTestB.StepName:='103 - Automaticky Rezim - kontrola stavu paletky';
            SC_P3_LeakageTestB.IdleTime.PT:= T#200ms;
            SC_P3_LeakageTestB.AlarmTime.PT:= T#5s;

            IF Paletka[i].PAR.TestovaciKus AND Paletka[i].PAR.CisloTestovacejStanice = 'ST_8A,8B' THEN
                IF P3_LeakageTestB.STAV.Tester_ON THEN
                    TestovaciKus:= TRUE;
                    SC_P3_LeakageTestB.ResetStep:= TRUE;
                    SC_P3_LeakageTestB.Step:= 113;
                ELSE
                    SC_P3_LeakageTestB.ResetStep:= TRUE;
                    SC_P3_LeakageTestB.Step:= 560;
                END_IF
            ELSIF Paletka[i].PAR.TestovaciKus AND Paletka[i].PAR.CisloTestovacejStanice <> 'ST_8A,8B' THEN
                SC_P3_LeakageTestB.ResetStep:= TRUE;
                SC_P3_LeakageTestB.Step:= 560;
            ELSIF Paletka[i].PAR.RevorkovyKus AND Paletka[i].PAR.CisloRevorkovejStanice = 'ST_8A,8B' THEN
                IF P3_LeakageTestB.STAV.Tester_ON THEN
                    Revork:= TRUE;
                    SC_P3_LeakageTestB.ResetStep:= TRUE;
                    SC_P3_LeakageTestB.Step:= 105;
                ELSE
                    SC_P3_LeakageTestB.ResetStep:= TRUE;
                    SC_P3_LeakageTestB.Step:= 560;
                END_IF
            ELSIF Paletka[i].PAR.RevorkovyKus AND Paletka[i].PAR.CisloRevorkovejStanice <> 'ST_8A,8B' THEN
                Revork:= FALSE;
                SC_P3_LeakageTestB.ResetStep:= TRUE;
                SC_P3_LeakageTestB.Step:= 560;
            ELSIF Paletka[i].PAR.StavPaletky = 'OK' AND P3_LeakageTestB.STAV.Tester_ON THEN
                SC_P3_LeakageTestB.ResetStep:= TRUE;
                SC_P3_LeakageTestB.Step:= 105;
            ELSIF Paletka[i].PAR.StavPaletky = 'OK' AND NOT P3_LeakageTestB.STAV.Tester_ON THEN
                SC_P3_LeakageTestB.ResetStep:= TRUE;
                SC_P3_LeakageTestB.Step:= 560;
            ELSIF Paletka[i].PAR.StavPaletky = 'NG' THEN
                SC_P3_LeakageTestB.ResetStep:= TRUE;
                SC_P3_LeakageTestB.Step:= 560;
            END_IF

        105:
            SC_P3_LeakageTestB.StepName:='105 - Automaticky Rezim - kontrola ukoncenia leakage testu';
            SC_P3_LeakageTestB.IdleTime.PT:= T#200ms;
            SC_P3_LeakageTestB.AlarmTime.PT:= T#5s;

            IF Paletka[i].VnutornyStav.LeakageTest_Ukonceny THEN
                SC_P3_LeakageTestB.ResetStep:= TRUE;
                SC_P3_LeakageTestB.Step:= 560;
            ELSE
                SC_P3_LeakageTestB.ResetStep:= TRUE;
                SC_P3_LeakageTestB.Step:= 110;
            END_IF

        110:
            SC_P3_LeakageTestB.StepName:='110 - Automaticky Rezim - cakam na prichod paletky na stanicu A a spustenie testovania';
            SC_P3_LeakageTestB.IdleTime.PT:= T#5s;
            SC_P3_LeakageTestB.AlarmTime.PT:= T#1M;
            SC_P3_LeakageTestB.AlarmTime.IN:= TRUE;

            IF NOT P3_StoperSrobovania.IN.PritomnostPaletky_S22 AND
                NOT P3_AkumulacnyStoper.IN.PritomnPaletky_IS65 AND
                NOT P3_LeakageTestA.IN.PritomnostPaletky_S23 THEN
                SC_P3_LeakageTestB.IdleTime.IN:= TRUE;
            ELSE
                SC_P3_LeakageTestB.IdleTime.IN:= FALSE;
            END_IF

            (*SC_P3_LeakageTestB.IdleTime.IN:= NOT P3_LeakageTestA.IN.PritomnostPaletky_S23;*)

            IF P3_LeakageTestB.KoniecCyklu THEN
                SC_P3_LeakageTestB.ResetStep:= TRUE;
                SC_P3_LeakageTestB.Step:= 113;
            ELSIF SC_P3_LeakageTestA.Step = 110 AND P3_LeakageTestA.IN.PritomnostPaletky_S23 THEN
                P3_LeakageTestB.OUT.KOM_StanicaA_StartTestovania:= TRUE;
                SC_P3_LeakageTestB.ResetStep:= TRUE;
                SC_P3_LeakageTestB.Step:= 113;
            ELSIF SC_P3_LeakageTestA.Step = 560 AND P3_LeakageTestA.IN.PritomnostPaletky_S23 THEN
                SC_P3_LeakageTestB.ResetStep:= TRUE;
                SC_P3_LeakageTestB.Step:= 113;
            ELSIF NOT P3_LeakageTestA.STAV.Tester_ON THEN
                SC_P3_LeakageTestB.ResetStep:= TRUE;
                SC_P3_LeakageTestB.Step:= 113;
            ELSIF SC_P3_LeakageTestB.IdleTime.Q THEN
                SC_P3_LeakageTestB.ResetStep:= TRUE;
                SC_P3_LeakageTestB.Step:= 113;
            ELSIF SC_P3_LeakageTestB.AlarmTime.Q THEN
                SC_P3_LeakageTestB.ResetStep:= TRUE;
                SC_P3_LeakageTestB.Step:= 113;
            END_IF

        113:
            SC_P3_LeakageTestB.StepName:='113 - Automaticky Rezim - vyziadanie stavu paletky zo servera, zacentrovanie paletky';
            SC_P3_LeakageTestB.IdleTime.PT:= T#200ms;
            SC_P3_LeakageTestB.AlarmTime.PT:= T#5s;
            SC_P3_LeakageTestB.IdleTime.IN:= TRUE;

            IF NOT SC_P3_LeakageTestB.Switch1 THEN
                TRCB_P3_LeakageTestB_ST8B.CMD.VyziadajStavPaletky_TYP1:= TRUE;
                Centrovacku_VYSUN:= TRUE;
                SC_P3_LeakageTestB.Switch1:= TRUE;
            END_IF

            IF TRCB_P3_LeakageTestB_ST8B.STATUS.KomunikaciaUkoncena THEN
                TRCB_P3_LeakageTestB_ST8B.CMD.VyziadajStavPaletky_TYP1:= FALSE;
                SC_P3_LeakageTestB.ResetStep:= TRUE;
                SC_P3_LeakageTestB.Step:= 114;
            ELSIF TRCB_P3_LeakageTestB_ST8B.STATUS.KomunikaciaError THEN
                TRCB_P3_LeakageTestB_ST8B.CMD.VyziadajStavPaletky_TYP1:= FALSE;
                SC_P3_LeakageTestB.ResetStep:= TRUE;
                SC_P3_LeakageTestB.Step:= 115;
            END_IF

        114:
            SC_P3_LeakageTestB.StepName:='114 - Automaticky Rezim - kontrola odpovede servera';
            SC_P3_LeakageTestB.IdleTime.PT:= T#200ms;
            SC_P3_LeakageTestB.AlarmTime.PT:= T#5s;

            IF NOT TRCB_P3_LeakageTestB_ST8B.STATUS.KomunikaciaUkoncena AND P3_LeakageTestB.IN.Centrovanie_VYSUNUTE_IS73 THEN
                IF TRCB_P3_LeakageTestB_ST8B.OUTPUTS.PovolenieCinnostiNaPaletke = 'OK' THEN
                    Paletka[i].VnutornyStav.KomunikaciaOtvorena:= TRUE;
                    IF TRCB_P3_LeakageTestB_ST8B.OUTPUTS.DruhCinnostiNaPaletke  = 'PRD;ST8B' THEN
                        SC_P3_LeakageTestB.ResetStep:= TRUE;
                        SC_P3_LeakageTestB.Step:= 118;
                    ELSIF TRCB_P3_LeakageTestB_ST8B.OUTPUTS.DruhCinnostiNaPaletke  = 'PRD;ST8A,ST8B' THEN
                        SC_P3_LeakageTestB.ResetStep:= TRUE;
                        SC_P3_LeakageTestB.Step:= 118;
                    ELSIF TRCB_P3_LeakageTestB_ST8B.OUTPUTS.DruhCinnostiNaPaletke  = 'SMP;ST8A,ST8B' THEN
                        SC_P3_LeakageTestB.ResetStep:= TRUE;
                        SC_P3_LeakageTestB.Step:= 118;
                    ELSE
                        Paletka[i].PAR.StavPaletky := 'NG';
                        SC_P3_LeakageTestB.ResetStep:= TRUE;
                        SC_P3_LeakageTestB.Step:= 116;
                    END_IF
                ELSIF TRCB_P3_LeakageTestB_ST8B.OUTPUTS.PovolenieCinnostiNaPaletke = 'NG' THEN
                    SC_P3_LeakageTestB.ResetStep:= TRUE;
                    SC_P3_LeakageTestB.Step:= 115;
                END_IF
            END_IF

        115:
            SC_P3_LeakageTestB.StepName:='115 - Automaticky Rezim - rozhodnutie obsluhy po odpovedi panatrace NG';
            SC_P3_LeakageTestB.IdleTime.PT:= T#200ms;
            SC_P3_LeakageTestB.AlarmTime.PT:= T#5s;

            P34_Vizu.ZobrazHL2_ST8:= TRUE;

            IF TRCB_P3_LeakTestB_OpatovnyDopyt THEN
                TRCB_P3_LeakTestB_OpatovnyDopyt:= FALSE;
                P34_Vizu.ZobrazHL2_ST8:= FALSE;
                SC_P3_LeakageTestB.ResetStep:= TRUE;
                SC_P3_LeakageTestB.Step:= 113;
            ELSIF TRCB_P3_LeakTestB_PaletkaNG THEN
                TRCB_P3_LeakTestB_PaletkaNG:= FALSE;
                P34_Vizu.ZobrazHL2_ST8:= FALSE;
                Paletka[i].PAR.StavPaletky := 'NG';
                SC_P3_LeakageTestB.ResetStep:= TRUE;
                SC_P3_LeakageTestB.Step:= 116;
            END_IF

        116:
            SC_P3_LeakageTestB.StepName:='116 - Automaticky Rezim - odcentrovanie paletky po odpovedi servera NG';
            SC_P3_LeakageTestB.IdleTime.PT:= T#200ms;
            SC_P3_LeakageTestB.AlarmTime.PT:= T#5s;

            IF NOT SC_P3_LeakageTestB.Switch1 THEN
                Centrovacku_ZASUN:= TRUE;
                SC_P3_LeakageTestB.Switch1:= TRUE;
            END_IF

            IF P3_LeakageTestB.IN.Centrovanie_ZASUNUTE_IS74 THEN
                SC_P3_LeakageTestB.ResetStep:= TRUE;
                SC_P3_LeakageTestB.Step:= 560;
            END_IF

        118:
            SC_P3_LeakageTestB.StepName:='118 - Automaticky Rezim - zacentrovanie paletky';
            SC_P3_LeakageTestB.IdleTime.PT:= T#200ms;
            SC_P3_LeakageTestB.AlarmTime.PT:= T#5s;

            IF NOT SC_P3_LeakageTestB.Switch1 THEN
                Centrovacku_VYSUN:= TRUE;
                SC_P3_LeakageTestB.Switch1:= TRUE;
            END_IF

            IF P3_LeakageTestB.IN.Centrovanie_VYSUNUTE_IS73 THEN
                SC_P3_LeakageTestB.ResetStep:= TRUE;
                SC_P3_LeakageTestB.Step:= 120;
            END_IF

        120:
            SC_P3_LeakageTestB.StepName:='120 - Automaticky Rezim - vysunutie horneho pritlaku';
            SC_P3_LeakageTestB.IdleTime.PT:= T#3s;
            SC_P3_LeakageTestB.AlarmTime.PT:= T#5s;

            IF NOT SC_P3_LeakageTestB.Switch1 THEN
                P3_LeakageTestB.OUT.PneuZamok_ODOMKNI_YV160:= TRUE;
                Pritlak_VYSUN:= TRUE;
                SC_P3_LeakageTestB.Switch1:= TRUE;
            END_IF

            IF P3_LeakageTestB.IN.Pritlak_VYSUNUTY_MS49 THEN
                SC_P3_LeakageTestB.ResetStep:= TRUE;
                SC_P3_LeakageTestB.Step:= 123;
            END_IF

        123:
            SC_P3_LeakageTestB.StepName:='123 - Automaticky Rezim - vysunutie spodneho kopita';
            SC_P3_LeakageTestB.IdleTime.PT:= T#1s;
            SC_P3_LeakageTestB.AlarmTime.PT:= T#5s;

            IF P3_LeakageTestB.IN.PritomnostKopita_IS69 AND P3_LeakageTestB.IN.Kopito_ZASUNUTE_IS70 THEN
                P3_LeakageTestB.OUT.Kopito_ZASUN_YV146:= FALSE;
                P3_LeakageTestB.OUT.Kopito_VYSUN_YV145:= TRUE;
                SC_P3_LeakageTestB.ResetStep:= TRUE;
                SC_P3_LeakageTestB.Step:= 125;
            END_IF

        125:
            SC_P3_LeakageTestB.StepName:='125 - Automaticky Rezim - cakam na spustenie testera';
            SC_P3_LeakageTestB.IdleTime.PT:= T#200ms;
            SC_P3_LeakageTestB.AlarmTime.PT:= T#5s;

            SC_P3_LeakageTestB.IdleTime.IN:= NOT P3_LeakageTestB.IN.Kopito_ZASUNUTE_IS70;

            IF SC_P3_LeakageTestB.IdleTime.Q  THEN
                SC_P3_LeakageTestB.ResetStep:= TRUE;
                SC_P3_LeakageTestB.Step:= 130;
            END_IF

        130:
            SC_P3_LeakageTestB.StepName:='130 - Automaticky Rezim - spustenie testera';
            SC_P3_LeakageTestB.IdleTime.PT:= T#4s800ms;
            SC_P3_LeakageTestB.AlarmTime.PT:= T#5s;

            IF NOT SC_P3_LeakageTestB.Switch1 AND AteqLeakageTester_B.Stav_READY THEN
                AteqLeakageTester_B.START_Testovania:= TRUE;
                Paletka[i].VnutornyStav.CinnostSpustena:= TRUE;
                SC_P3_LeakageTestB.IdleTime.IN:= TRUE;
                SC_P3_LeakageTestB.Switch1:= TRUE;
            END_IF

            IF NOT AteqLeakageTester_B.Stav_READY AND AteqLeakageTester_B.Stav_START_DONE AND NOT AteqLeakageTester_B.VysledokTestovania_OK AND NOT AteqLeakageTester_B.VysledokTestovania_NG AND SC_P3_LeakageTestB.IdleTime.Q THEN
                P3_LeakageTestB.OUT.PneuZamok_ODOMKNI_YV160:= FALSE;
                P3_LeakageTestB.OUT.Pritlak_VYSUN_YV161:= FALSE;
                SC_P3_LeakageTestB.ResetStep:= TRUE;
                SC_P3_LeakageTestB.Step:= 133;
            END_IF

        133:
            SC_P3_LeakageTestB.StepName:='130 - Automaticky Rezim - nacitanie parametrov testera';
            SC_P3_LeakageTestB.IdleTime.PT:= T#500ms;
            SC_P3_LeakageTestB.AlarmTime.PT:= T#5s;

            IF AteqLeakageTester_B.Stav_READY THEN
                AteqLeakageTester_B.START_Testovania:= FALSE;
                AteqLeakageTester_B.CitajParametreTestera:= TRUE;
            END_IF

            SC_P3_LeakageTestB.IdleTime.IN:= AteqLeakageTester_B.Stav_CitanieParametrov_OK;

            IF AteqLeakageTester_B.Stav_CitanieParametrov_OK AND SC_P3_LeakageTestB.IdleTime.Q THEN
                Reports.LeakageTest.CasPlnenia.StanicaB:= REAL_TO_STRING(AteqLeakageTester_B.CasPnenia);
                Reports.LeakageTest.CasStabilizacie.StanicaB:= REAL_TO_STRING(AteqLeakageTester_B.CasStabilizacie);
                Reports.LeakageTest.TlakPlnenia.StanicaB:= REAL_TO_STRING(AteqLeakageTester_B.TlakPlnenia);
                Reports.LeakageTest.ToleranciaPritlaku_MIN.StanicaB:= '';
                Reports.LeakageTest.ToleranciaPritlaku_MAX.StanicaB:= '';
                Reports.LeakageTest.TlakPritlaku.StanicaB:= REAL_TO_STRING(P3_LeakageTestB.IN.PreratanyVyrovnavaciTlak_Bar);
                Reports.LeakageTest.TlakUniku.StanicaB:= REAL_TO_STRING(AteqLeakageTester_B.TlakUniku);
                Reports.LeakageTest.ToleranciaTlakUniku_MIN.StanicaB:= REAL_TO_STRING(AteqLeakageTester_B.Tolerancia * -1);
                Reports.LeakageTest.ToleranciaTlakUniku_MAX.StanicaB:= REAL_TO_STRING(AteqLeakageTester_B.Tolerancia);
                Reports.LeakageTest.Tolerancia.StanicaB:= REAL_TO_STRING(AteqLeakageTester_B.Tolerancia);
                AteqLeakageTester_B.CitajParametreTestera:= FALSE;
                SC_P3_LeakageTestB.ResetStep:= TRUE;
                SC_P3_LeakageTestB.Step:= 135;
            END_IF

        135:
            SC_P3_LeakageTestB.StepName:='135 - Automaticky Rezim - kontrola výsledku testu';
            SC_P3_LeakageTestB.IdleTime.PT:= T#1s;
            SC_P3_LeakageTestB.AlarmTime.PT:= T#5s;

            IF AteqLeakageTester_B.VysledokTestovania_OK THEN
                Paletka[i].VnutornyStav.LeakageTest_Ukonceny:= TRUE;
                Paletka[i].PAR.StavPowerCP:= 'PASS';
                Reports.LeakageTest.VyslednyReport.StanicaB:= 'PASS';
                Paletka[i].VnutornyStav.CinnostUkoncena:= TRUE;
                SC_P3_LeakageTestB.ResetStep:= TRUE;
                SC_P3_LeakageTestB.Step:= 140;
            ELSE
                IF NOT Revork THEN
                    OpakovanyTest:= TRUE;
                END_IF
                Paletka[i].PAR.StavPowerCP:= 'FAIL';
                Paletka[i].VnutornyStav.CinnostUkoncena:= TRUE;
                Reports.LeakageTest.VyslednyReport.StanicaB:= 'FAIL';
                SC_P3_LeakageTestB.ResetStep:= TRUE;
                SC_P3_LeakageTestB.Step:= 140;
            END_IF

        140:
            SC_P3_LeakageTestB.StepName:='140 - Automaticky Rezim - cakam na ukoncenie testovania testera stanice A';
            SC_P3_LeakageTestB.IdleTime.PT:= T#1s;
            SC_P3_LeakageTestB.AlarmTime.PT:= T#5s;

            IF NOT AteqLeakageTester_A.START_Testovania THEN
                SC_P3_LeakageTestB.ResetStep:= TRUE;
                SC_P3_LeakageTestB.Step:= 150;
            ELSIF P3_LeakageTestB.RR_TestovaciaSekvencia THEN
                SC_P3_LeakageTestB.ResetStep:= TRUE;
                SC_P3_LeakageTestB.Step:= 150;
            END_IF

        150:
            SC_P3_LeakageTestB.StepName:='150 - Automaticky Rezim - zasunutie spodneho kopita';
            SC_P3_LeakageTestB.IdleTime.PT:= T#200ms;
            SC_P3_LeakageTestB.AlarmTime.PT:= T#5s;

            P3_LeakageTestB.OUT.Kopito_VYSUN_YV145:= FALSE;
            P3_LeakageTestB.OUT.Kopito_ZASUN_YV146:= TRUE;

            IF P3_LeakageTestB.IN.Kopito_ZASUNUTE_IS70 THEN
                SC_P3_LeakageTestB.ResetStep:= TRUE;
                SC_P3_LeakageTestB.Step:= 153;
            END_IF

        153:
            SC_P3_LeakageTestB.StepName:='153 - Automaticky Rezim - zasunutie horneho pritlaku';
            SC_P3_LeakageTestB.IdleTime.PT:= T#200ms;
            SC_P3_LeakageTestB.AlarmTime.PT:= T#5s;

            IF NOT SC_P3_LeakageTestB.Switch1 THEN
                P3_LeakageTestB.OUT.PneuZamok_ODOMKNI_YV160:= TRUE;
                Pritlak_ZASUN:= TRUE;
                SC_P3_LeakageTestB.IdleTime.IN:= TRUE;
                SC_P3_LeakageTestB.Switch1:= TRUE;
            END_IF

            IF SC_P3_LeakageTestB.IdleTime.Q THEN
                SC_P3_LeakageTestB.ResetStep:= TRUE;
                SC_P3_LeakageTestB.Step:= 545;
            END_IF

            //Odcentrovanie paletky//

        545:
            SC_P3_LeakageTestB.StepName:='545 - Automaticky Rezim - odcentrovanie paletky';
            SC_P3_LeakageTestB.IdleTime.PT:= T#200ms;
            SC_P3_LeakageTestB.AlarmTime.PT:= T#5s;

            Centrovacku_ZASUN:= TRUE;
            IF P3_LeakageTestB.RR_TestovaciaSekvencia THEN
                SC_P3_LeakageTestB.ResetStep:= TRUE;
                SC_P3_LeakageTestB.Step:= 558;
            ELSE
                SC_P3_LeakageTestB.ResetStep:= TRUE;
                SC_P3_LeakageTestB.Step:= 550;
            END_IF

            //Odoslanie dát na server//

        550:
            SC_P3_LeakageTestB.StepName:='550 - Automaticky Rezim - odoslanie stavu paletky na server';
            SC_P3_LeakageTestB.IdleTime.PT:= T#200ms;
            SC_P3_LeakageTestB.AlarmTime.PT:= T#5s;

            IF NOT SC_P3_LeakageTestB.Switch1 THEN
                TRCB_P3_LeakageTestB_ST8B.CMD.OdosliStavPaletky_TYP2:= TRUE;
                SC_P3_LeakageTestB.Switch1:= TRUE;
            END_IF

            IF TRCB_P3_LeakageTestB_ST8B.STATUS.KomunikaciaUkoncena THEN
                TRCB_P3_LeakageTestB_ST8B.CMD.OdosliStavPaletky_TYP2:= FALSE;
                SC_P3_LeakageTestB.ResetStep:= TRUE;
                SC_P3_LeakageTestB.Step:= 553;
            ELSIF TRCB_P3_LeakageTestB_ST8B.STATUS.KomunikaciaError THEN
                //                P34_Alarmy[313]:= TRUE;
                //                P3_PoruchaST3:= TRUE;
            END_IF

        553:
            SC_P3_LeakageTestB.StepName:='553 - Automaticky Rezim - kontrola odpovede servera';
            SC_P3_LeakageTestB.IdleTime.PT:= T#200ms;
            SC_P3_LeakageTestB.AlarmTime.PT:= T#5s;

            IF NOT TRCB_P3_LeakageTestB_ST8B.STATUS.KomunikaciaUkoncena THEN
                IF TRCB_P3_LeakageTestB_ST8B.OUTPUTS.PovolenieCinnostiNaPaletke = 'OK' THEN
                    Paletka[i].PAR.StavPaletky:= 'OK';
                    SC_P3_LeakageTestB.ResetStep:= TRUE;
                    SC_P3_LeakageTestB.Step:= 554;
                ELSIF TRCB_P3_LeakageTestB_ST8B.OUTPUTS.PovolenieCinnostiNaPaletke = 'NG' THEN
                    Paletka[i].PAR.StavPaletky:= 'NG';
                    SC_P3_LeakageTestB.ResetStep:= TRUE;
                    SC_P3_LeakageTestB.Step:= 554;
                END_IF
            END_IF

        554:
            SC_P3_LeakageTestB.StepName:='554 - Automaticky Rezim - kontrola poctu testovani';
            SC_P3_LeakageTestB.IdleTime.PT:= T#1s;
            SC_P3_LeakageTestB.AlarmTime.PT:= T#5s;
            SC_P3_LeakageTestB.IdleTime.IN:= TRUE;

            IF NOT SC_P3_LeakageTestB.Switch1 THEN
                PocetOpakovaniTestu:= PocetOpakovaniTestu + 1;
                SC_P3_LeakageTestB.Switch1:= TRUE;
            END_IF

            IF OpakovanyTest AND PocetOpakovaniTestu < 2 AND SC_P3_LeakageTestB.IdleTime.Q AND NOT TestovaciKus THEN
                OpakovanyTest:= FALSE;
                SC_P3_LeakageTestB.ResetStep:= TRUE;
                SC_P3_LeakageTestB.Step:= 113;
            ELSIF OpakovanyTest AND PocetOpakovaniTestu >= 2 AND NOT TestovaciKus THEN
                Paletka[i].VnutornyStav.LeakageTest_Ukonceny:= TRUE;
                OpakovanyTest:= FALSE;
                PocetOpakovaniTestu:= 0;
                SC_P3_LeakageTestB.ResetStep:= TRUE;
                SC_P3_LeakageTestB.Step:= 555;
            ELSIF NOT OpakovanyTest OR TestovaciKus THEN
                SC_P3_LeakageTestB.ResetStep:= TRUE;
                SC_P3_LeakageTestB.Step:= 555;
            END_IF

        555:
            SC_P3_LeakageTestB.StepName:='555 - Automaticky Rezim - vyhodnotenie stavu paletky';
            SC_P3_LeakageTestB.IdleTime.PT:= T#200ms;
            SC_P3_LeakageTestB.AlarmTime.PT:= T#5s;

            IF Paletka[i].PAR.StavPaletky = 'OK' THEN
                IF Paletka[i].PAR.StavPowerCP = 'PASS' THEN
                    Paletka[i].PAR.StavPaletky:= 'OK';
                ELSIF Paletka[i].PAR.StavPowerCP = 'FAIL' THEN
                    Paletka[i].PAR.StavPaletky:= 'NG';
                END_IF
            END_IF
            Paletka[i].VnutornyStav.KomunikaciaUzavreta:= TRUE;

            SC_P3_LeakageTestB.ResetStep:= TRUE;
            SC_P3_LeakageTestB.Step:= 558;

        558:
            SC_P3_LeakageTestB.StepName:='558 - Automaticky Rezim - kontrola otvorenia testera';
            SC_P3_LeakageTestB.IdleTime.PT:= T#200ms;
            SC_P3_LeakageTestB.AlarmTime.PT:= T#5s;

            IF P3_LeakageTestB.IN.Centrovanie_ZASUNUTE_IS74 AND P3_LeakageTestB.IN.Pritlak_ZASUNUTY_MS48 AND P3_LeakageTestB.IN.Kopito_ZASUNUTE_IS70 THEN
                P3_LeakageTestB.OUT.PneuZamok_ODOMKNI_YV160:= FALSE;
                IF P3_LeakageTestB.RR_TestovaciaSekvencia THEN
                    P3_LeakageTestB.RR_TestovaciaSekvencia:= FALSE;
                    SC_P3_LeakageTestB.ResetStep:= TRUE;
                    SC_P3_LeakageTestB.Step:= 700;
                ELSE
                    SC_P3_LeakageTestB.ResetStep:= TRUE;
                    SC_P3_LeakageTestB.Step:= 560;
                END_IF
            END_IF

            //Vyvezenie paletky//

        560:
            SC_P3_LeakageTestB.StepName:='560 - Automaticky Rezim - cakam na vyvezenie na stoper funkcneho testu A';
            SC_P3_LeakageTestB.IdleTime.PT:= T#200ms;
            SC_P3_LeakageTestB.AlarmTime.PT:= T#5s;

            IF P3_LeakageTestB.KoniecCyklu THEN
                SC_P3_LeakageTestB.ResetStep:= TRUE;
                SC_P3_LeakageTestB.Step:= 0;
            ELSIF ((NOT P4_FunkcnyTestA.IN.PritomnostPaletky_S10 AND SC_P4_FunkcnyTestA.Step = 100) OR (P4_FunkcnyTestA.OUT.ZasunStoper_YV163 AND SC_P4_FunkcnyTestA.Step = 561)) AND NOT P3_LeakageTestB.STAV.PrebiehaVyvezeniePaletky AND NOT TEST THEN
                P3_LeakageTestB.OUT.ZasunStoper_YV135:= TRUE;
                P3_LeakageTestB.STAV.PrebiehaVyvezeniePaletky:= TRUE;
                SC_P3_LeakageTestB.ResetStep:= TRUE;
                SC_P3_LeakageTestB.Step:= 561;
            END_IF

        561:
            SC_P3_LeakageTestB.StepName:='561 - Automaticky Rezim - ukoncenie vyvazania na stoper funkcneho testu A';
            SC_P3_LeakageTestB.IdleTime.PT:= T#200ms;
            SC_P3_LeakageTestB.AlarmTime.PT:= T#10s;

            SC_P3_LeakageTestB.IdleTime.IN:= NOT P3_LeakageTestB.IN.PritomnostPaletky_S24;
            SC_P3_LeakageTestB.AlarmTime.IN:= P3_LeakageTestB.IN.PritomnostPaletky_S24;

            IF NOT P3_LeakageTestB.IN.PritomnostPaletky_S24 THEN
                IF Revork THEN
                    Paletka[i].PAR.RevorkovyKus:= FALSE;
                    Paletka[i].PAR.CisloRevorkovejStanice:= '';
                    Revork:= FALSE;
                END_IF
                P3_LeakageTestB.OUT.ZasunStoper_YV135:= FALSE;
                TestovaciKus:= FALSE;
                OpakovanyTest:= FALSE;
                PocetOpakovaniTestu:= 0;
                Paletka[i].PAR.StavPowerCP:= '';
                Paletka[i].VnutornyStav.CinnostSpustena:= FALSE;
                Paletka[i].VnutornyStav.CinnostUkoncena:= FALSE;
                Paletka[i].VnutornyStav.FotkyOdoslane:= FALSE;
                Paletka[i].VnutornyStav.KomunikaciaOtvorena:= FALSE;
                Paletka[i].VnutornyStav.KomunikaciaUzavreta:= FALSE;
                Reports.LeakageTest.CasPlnenia.StanicaB:= '';
                Reports.LeakageTest.VyslednyReport.StanicaB:= '';
                Reports.LeakageTest.CasStabilizacie.StanicaB:= '';
                Reports.LeakageTest.TlakPlnenia.StanicaB:= '';
                Reports.LeakageTest.ToleranciaPritlaku_MIN.StanicaB:= '';
                Reports.LeakageTest.ToleranciaPritlaku_MAX.StanicaB:= '';
                Reports.LeakageTest.TlakPritlaku.StanicaB:= '';
                Reports.LeakageTest.TlakUniku.StanicaB:= '';
                Reports.LeakageTest.Tolerancia.StanicaB:= '';
            END_IF

            IF SC_P3_LeakageTestB.IdleTime.Q AND NOT P3_LeakageTestB.OUT.ZasunStoper_YV135 THEN
                SC_P3_LeakageTestB.ResetStep:= TRUE;
                SC_P3_LeakageTestB.Step:= 100;
            ELSIF SC_P3_LeakageTestB.AlarmTime.Q THEN
                P34_Alarmy[358]:= TRUE;
                P3_Pracovisko.KoniecCyklu:= TRUE;
                SC_P3_LeakageTestB.ResetStep:= TRUE;
                SC_P3_LeakageTestB.Step:= 0;
            END_IF

            //*******************************************************Manuálny režim*******************************************************************************//
        700:
            SC_P3_LeakageTestB.StepName:='700 - Manualny Rezim';
            SC_P3_LeakageTestB.IdleTime.PT:= T#8s;
            SC_P3_LeakageTestB.AlarmTime.PT:= T#5s;

            P3_LeakageTestB.OUT.PneuZamok_ODOMKNI_YV160:= TRUE;

            //Vysunutie spodného kopita//
            IF P3_LeakageTestB.RR_VysunSpodneKopito THEN
                P3_LeakageTestB.OUT.Kopito_ZASUN_YV146:= FALSE;
                P3_LeakageTestB.OUT.Kopito_VYSUN_YV145:= TRUE;
            ELSE
                P3_LeakageTestB.OUT.Kopito_VYSUN_YV145:= FALSE;
                P3_LeakageTestB.OUT.Kopito_ZASUN_YV146:= TRUE;
            END_IF

            //Spustenie testovacej sekvencie//
            P3_LeakageTestB.STAV.TestovaciaSekvencia_BUSY:= P3_LeakageTestB.RR_TestovaciaSekvencia;

            IF P3_LeakageTestB.RR_TestovaciaSekvencia THEN
                IF P3_LeakageTestB.IN.PritomnostPaletky_S24 THEN
                    SC_P3_LeakageTestB.ResetStep:= TRUE;
                    SC_P3_LeakageTestB.Step:= 118;
                ELSE
                    P3_LeakageTestB.RR_TestovaciaSekvencia:= FALSE;
                END_IF
            END_IF

    END_CASE

END_PROGRAM

PROGRAM _EXIT
	(* Insert code here *)

END_PROGRAM
```

#### Variables.var - Local variables
```iecst
VAR
	SC_OvlCentrovacky : SequenceControlTyp;
	Centrovacku_VYSUN : BOOL;
	Centrovacku_ZASUN : BOOL;
	PrecitaneCisloPaletky : STRING[3];
	ServerOdpoved_StavPowerCP : STRING[5];
	i : USINT;
	SC_OvlPritlaku : SequenceControlTyp;
	Pritlak_VYSUN : BOOL;
	Pritlak_ZASUN : BOOL;
	TEST : BOOL;
	PocetDopytovNaServer : USINT;
	CasPneniaREAL : REAL;
	TlakPlneniaREAL : REAL;
	ToleranciaREAL : REAL;
	CasStabilizacieREAL : REAL;
	TlakUnikuREAL : REAL;
	TestovaciKus : BOOL;
	Revork : BOOL;
	Triger_0 : BOOL;
	Triger_1 : BOOL;
	PocetOpakovaniTestu : USINT;
	OpakovanyTest : BOOL;
END_VAR
```

#### IOLinkKomunikacia.st
```iecst
ACTION IOLinkKomunikacia:

	//Snímač paletky//
	P3_LeakageTestB.IN.PritomnostPaletky_S24:= P3_LeakageTestB.PAR.SnimacPaletky_IOLinkInputs[1].0;
	P3_LeakageTestB.IN.PrecitaneCisloPaletky_S24:= P3_LeakageTestB.PAR.SnimacPaletky_IOLinkInputs[9];

	//Snímač tlaku//
	P3_LeakageTestB.IN.VyrovnavaciTlak_OK_S27:= P3_LeakageTestB.PAR.SnimacTlaku_IOLinkInputs.0;

	P3_LeakageTestB.IN.PrecitanyVyrovnavaciTlak_S27.0:= P3_LeakageTestB.PAR.SnimacTlaku_IOLinkInputs.2;
	P3_LeakageTestB.IN.PrecitanyVyrovnavaciTlak_S27.1:= P3_LeakageTestB.PAR.SnimacTlaku_IOLinkInputs.3;
	P3_LeakageTestB.IN.PrecitanyVyrovnavaciTlak_S27.2:= P3_LeakageTestB.PAR.SnimacTlaku_IOLinkInputs.4;
	P3_LeakageTestB.IN.PrecitanyVyrovnavaciTlak_S27.3:= P3_LeakageTestB.PAR.SnimacTlaku_IOLinkInputs.5;
	P3_LeakageTestB.IN.PrecitanyVyrovnavaciTlak_S27.4:= P3_LeakageTestB.PAR.SnimacTlaku_IOLinkInputs.6;
	P3_LeakageTestB.IN.PrecitanyVyrovnavaciTlak_S27.5:= P3_LeakageTestB.PAR.SnimacTlaku_IOLinkInputs.7;
	P3_LeakageTestB.IN.PrecitanyVyrovnavaciTlak_S27.6:= P3_LeakageTestB.PAR.SnimacTlaku_IOLinkInputs.8;
	P3_LeakageTestB.IN.PrecitanyVyrovnavaciTlak_S27.7:= P3_LeakageTestB.PAR.SnimacTlaku_IOLinkInputs.9;
	P3_LeakageTestB.IN.PrecitanyVyrovnavaciTlak_S27.8:= P3_LeakageTestB.PAR.SnimacTlaku_IOLinkInputs.10;
	P3_LeakageTestB.IN.PrecitanyVyrovnavaciTlak_S27.9:= P3_LeakageTestB.PAR.SnimacTlaku_IOLinkInputs.11;
	P3_LeakageTestB.IN.PrecitanyVyrovnavaciTlak_S27.10:= P3_LeakageTestB.PAR.SnimacTlaku_IOLinkInputs.12;
	P3_LeakageTestB.IN.PrecitanyVyrovnavaciTlak_S27.11:= P3_LeakageTestB.PAR.SnimacTlaku_IOLinkInputs.13;
	P3_LeakageTestB.IN.PrecitanyVyrovnavaciTlak_S27.12:= P3_LeakageTestB.PAR.SnimacTlaku_IOLinkInputs.14;
	P3_LeakageTestB.IN.PrecitanyVyrovnavaciTlak_S27.13:= P3_LeakageTestB.PAR.SnimacTlaku_IOLinkInputs.15;

	P3_LeakageTestB.IN.PreratanyVyrovnavaciTlak_Bar:= P3_LeakageTestB.IN.PrecitanyVyrovnavaciTlak_S27 * 0.1;

END_ACTION
```

#### OvlCentrovacky.st
```iecst
ACTION OvlCentrovacky:

	//Volanie funkcie SequenceControl//
	SequenceControl(SC:= SC_OvlCentrovacky);

	CASE SC_OvlCentrovacky.Step OF

		0:
			SC_OvlCentrovacky.StepName:= '0 - Nulovanie';
			Centrovacku_VYSUN:= FALSE;
			Centrovacku_ZASUN:= FALSE;
			P3_LeakageTestB.OUT.VysunCentrovanie_YV147:= FALSE;
			P3_LeakageTestB.OUT.ZasunCentrovanie_YV148:= FALSE;

			IF SC_P3_LeakageTestB.Step <> 0 THEN
				SC_OvlCentrovacky.ResetStep:= TRUE;
				SC_OvlCentrovacky.Step:= 1;
			END_IF

		1:
			SC_OvlCentrovacky.StepName:= '1 - Rozhodnutie o cinnosti';
			IF Centrovacku_VYSUN THEN
				SC_OvlCentrovacky.Step:= 10;
			ELSIF Centrovacku_ZASUN THEN
				SC_OvlCentrovacky.Step:= 20;
			END_IF

		10:
			SC_OvlCentrovacky.StepName:= '10 - Vysunutie centrovacky';
			SC_OvlCentrovacky.IdleTime.PT:= T#3s;
			SC_OvlCentrovacky.AlarmTime.PT:= T#30s;

			IF P3_LeakageTestB.Automat THEN
				SC_OvlCentrovacky.AlarmTime.IN:= TRUE;
			ELSE
				SC_OvlCentrovacky.IdleTime.IN:= TRUE;
			END_IF

			IF NOT SC_OvlCentrovacky.Switch1 THEN
				P3_LeakageTestB.OUT.ZasunCentrovanie_YV148:= FALSE;
				P3_LeakageTestB.OUT.VysunCentrovanie_YV147:= TRUE;
				SC_OvlCentrovacky.Switch1:= TRUE;
			END_IF

            IF P3_LeakageTestB.IN.Centrovanie_VYSUNUTE_IS73 THEN
                SC_OvlCentrovacky.IdleTime.IN:= TRUE;
            END_IF

			IF SC_OvlCentrovacky.IdleTime.Q THEN
			    SC_OvlCentrovacky.ResetStep:= TRUE;
				SC_OvlCentrovacky.Step:= 0;
			ELSIF SC_OvlCentrovacky.AlarmTime.Q THEN
				P34_Alarmy[304]:= TRUE;
				P3_PoruchaST3:= TRUE;
			END_IF

		20:
			SC_OvlCentrovacky.StepName:= '20 - Zasunutie centrovacky';
			SC_OvlCentrovacky.IdleTime.PT:= T#3s;
			SC_OvlCentrovacky.AlarmTime.PT:= T#30s;

			IF P3_LeakageTestB.Automat THEN
				SC_OvlCentrovacky.AlarmTime.IN:= TRUE;
			ELSE
				SC_OvlCentrovacky.IdleTime.IN:= TRUE;
			END_IF

			IF NOT SC_OvlCentrovacky.Switch1 THEN
				P3_LeakageTestB.OUT.VysunCentrovanie_YV147:= FALSE;
				P3_LeakageTestB.OUT.ZasunCentrovanie_YV148:= TRUE;
				SC_OvlCentrovacky.Switch1:= TRUE;
			END_IF

			IF P3_LeakageTestB.IN.Centrovanie_ZASUNUTE_IS74 OR SC_OvlCentrovacky.IdleTime.Q THEN
				SC_OvlCentrovacky.ResetStep:= TRUE;
				SC_OvlCentrovacky.Step:= 0;
			ELSIF SC_OvlCentrovacky.AlarmTime.Q THEN
				P34_Alarmy[305]:= TRUE;
				P3_PoruchaST3:= TRUE;
			END_IF

	END_CASE

END_ACTION
```

#### OvlPritlaku.st
```iecst
ACTION OvlPritlaku:

	//Volanie funkcie SequenceControl//
	SequenceControl(SC:= SC_OvlPritlaku);

	CASE SC_OvlPritlaku.Step OF

		0:
			SC_OvlPritlaku.StepName:= '0 - Nulovanie';
			Pritlak_VYSUN:= FALSE;
			Pritlak_ZASUN:= FALSE;
			(*P3_LeakageTestB.OUT.Pritlak_VYSUN_YV161:= FALSE;*)
			P3_LeakageTestB.OUT.Pritlak_ZASUN_YV162:= FALSE;

			IF SC_P3_LeakageTestB.Step <> 0 THEN
				SC_OvlPritlaku.ResetStep:= TRUE;
				SC_OvlPritlaku.Step:= 1;
			END_IF

		1:
			SC_OvlPritlaku.StepName:= '1 - Rozhodnutie o cinnosti';
			IF Pritlak_VYSUN THEN
				SC_OvlPritlaku.Step:= 10;
			ELSIF Pritlak_ZASUN THEN
				SC_OvlPritlaku.Step:= 20;
			END_IF

		10:
			SC_OvlPritlaku.StepName:= '10 - Vysunutie pritlaku';
			SC_OvlPritlaku.IdleTime.PT:= T#3s;
			SC_OvlPritlaku.AlarmTime.PT:= T#30s;

			IF P3_LeakageTestB.Automat THEN
				SC_OvlPritlaku.AlarmTime.IN:= TRUE;
			ELSE
				SC_OvlPritlaku.IdleTime.IN:= TRUE;
			END_IF

			IF NOT SC_OvlPritlaku.Switch1 THEN
				P3_LeakageTestB.OUT.Pritlak_ZASUN_YV162:= FALSE;
				P3_LeakageTestB.OUT.Pritlak_VYSUN_YV161:= TRUE;
				SC_OvlPritlaku.Switch1:= TRUE;
			END_IF

			IF P3_LeakageTestB.IN.Pritlak_VYSUNUTY_MS49 OR SC_OvlPritlaku.IdleTime.Q THEN
				SC_OvlPritlaku.ResetStep:= TRUE;
				SC_OvlPritlaku.Step:= 0;
			ELSIF SC_OvlPritlaku.AlarmTime.Q THEN
				P34_Alarmy[308]:= TRUE;
				P3_PoruchaST3:= TRUE;
			END_IF

		20:
			SC_OvlPritlaku.StepName:= '20 - Zasunutie pritlaku';
			SC_OvlPritlaku.IdleTime.PT:= T#3s;
			SC_OvlPritlaku.AlarmTime.PT:= T#30s;

			IF P3_LeakageTestB.Automat THEN
				SC_OvlPritlaku.AlarmTime.IN:= TRUE;
			ELSE
				SC_OvlPritlaku.IdleTime.IN:= TRUE;
			END_IF

			IF NOT SC_OvlPritlaku.Switch1 THEN
				P3_LeakageTestB.OUT.Pritlak_VYSUN_YV161:= FALSE;
				P3_LeakageTestB.OUT.Pritlak_ZASUN_YV162:= TRUE;
				SC_OvlPritlaku.Switch1:= TRUE;
			END_IF

			IF P3_LeakageTestB.IN.Pritlak_ZASUNUTY_MS48 OR SC_OvlPritlaku.IdleTime.Q THEN
				SC_OvlPritlaku.ResetStep:= TRUE;
				SC_OvlPritlaku.Step:= 0;
			ELSIF SC_OvlPritlaku.AlarmTime.Q THEN
				P34_Alarmy[309]:= TRUE;
				P3_PoruchaST3:= TRUE;
			END_IF

	END_CASE

END_ACTION
```

#### TesterKomunikacia.st
```iecst
ACTION TesterKomunikacia:

	//Vstupy z Testera do PLC//
	AteqLeakageTester_B.Stav_RESET_DONE:= AteqLeakageTester_B.Profinet_PLC_INPUTS[1].0;
	AteqLeakageTester_B.Stav_START_DONE:= AteqLeakageTester_B.Profinet_PLC_INPUTS[1].1;
	AteqLeakageTester_B.Stav_ZmenaProgramu_DONE:= AteqLeakageTester_B.Profinet_PLC_INPUTS[1].3;
    AteqLeakageTester_B.Stav_CitanieParametrov_OK:= AteqLeakageTester_B.Profinet_PLC_INPUTS[1].5;

    AteqLeakageTester_B.Stav_CitanieParametrov_ERROR:= AteqLeakageTester_B.Profinet_PLC_INPUTS[3].5;

	AteqLeakageTester_B.CisloAktualnehoProgramu.0:= AteqLeakageTester_B.Profinet_PLC_INPUTS[7].0;
	AteqLeakageTester_B.CisloAktualnehoProgramu.1:= AteqLeakageTester_B.Profinet_PLC_INPUTS[7].1;
	AteqLeakageTester_B.CisloAktualnehoProgramu.2:= AteqLeakageTester_B.Profinet_PLC_INPUTS[7].2;
	AteqLeakageTester_B.CisloAktualnehoProgramu.3:= AteqLeakageTester_B.Profinet_PLC_INPUTS[7].3;
	AteqLeakageTester_B.CisloAktualnehoProgramu.4:= AteqLeakageTester_B.Profinet_PLC_INPUTS[7].4;
	AteqLeakageTester_B.CisloAktualnehoProgramu.5:= AteqLeakageTester_B.Profinet_PLC_INPUTS[7].5;
	AteqLeakageTester_B.CisloAktualnehoProgramu.6:= AteqLeakageTester_B.Profinet_PLC_INPUTS[7].6;
	AteqLeakageTester_B.CisloAktualnehoProgramu.7:= AteqLeakageTester_B.Profinet_PLC_INPUTS[7].7;

	AteqLeakageTester_B.CisloAktualnehoProgramu.8:= AteqLeakageTester_B.Profinet_PLC_INPUTS[8].0;
	AteqLeakageTester_B.CisloAktualnehoProgramu.9:= AteqLeakageTester_B.Profinet_PLC_INPUTS[8].1;
	AteqLeakageTester_B.CisloAktualnehoProgramu.10:= AteqLeakageTester_B.Profinet_PLC_INPUTS[8].2;
	AteqLeakageTester_B.CisloAktualnehoProgramu.11:= AteqLeakageTester_B.Profinet_PLC_INPUTS[8].3;
	AteqLeakageTester_B.CisloAktualnehoProgramu.12:= AteqLeakageTester_B.Profinet_PLC_INPUTS[8].4;
	AteqLeakageTester_B.CisloAktualnehoProgramu.13:= AteqLeakageTester_B.Profinet_PLC_INPUTS[8].5;
	AteqLeakageTester_B.CisloAktualnehoProgramu.14:= AteqLeakageTester_B.Profinet_PLC_INPUTS[8].6;
	AteqLeakageTester_B.CisloAktualnehoProgramu.15:= AteqLeakageTester_B.Profinet_PLC_INPUTS[8].7;

	AteqLeakageTester_B.VysledokTestovania_OK:= AteqLeakageTester_B.Profinet_PLC_INPUTS[13].0;
	AteqLeakageTester_B.VysledokTestovania_NG:= AteqLeakageTester_B.Profinet_PLC_INPUTS[13].1;
	AteqLeakageTester_B.Stav_ERROR:= AteqLeakageTester_B.Profinet_PLC_INPUTS[13].3;
	AteqLeakageTester_B.Stav_READY:= AteqLeakageTester_B.Profinet_PLC_INPUTS[13].5;

    AteqLeakageTester_B.ReadParameter_1.0:= AteqLeakageTester_B.Profinet_PLC_INPUTS[35].0;
    AteqLeakageTester_B.ReadParameter_1.1:= AteqLeakageTester_B.Profinet_PLC_INPUTS[35].1;
    AteqLeakageTester_B.ReadParameter_1.2:= AteqLeakageTester_B.Profinet_PLC_INPUTS[35].2;
    AteqLeakageTester_B.ReadParameter_1.3:= AteqLeakageTester_B.Profinet_PLC_INPUTS[35].3;
    AteqLeakageTester_B.ReadParameter_1.4:= AteqLeakageTester_B.Profinet_PLC_INPUTS[35].4;
    AteqLeakageTester_B.ReadParameter_1.5:= AteqLeakageTester_B.Profinet_PLC_INPUTS[35].5;
    AteqLeakageTester_B.ReadParameter_1.6:= AteqLeakageTester_B.Profinet_PLC_INPUTS[35].6;
    AteqLeakageTester_B.ReadParameter_1.7:= AteqLeakageTester_B.Profinet_PLC_INPUTS[35].7;
    AteqLeakageTester_B.ReadParameter_1.8:= AteqLeakageTester_B.Profinet_PLC_INPUTS[36].0;
    AteqLeakageTester_B.ReadParameter_1.9:= AteqLeakageTester_B.Profinet_PLC_INPUTS[36].1;
    AteqLeakageTester_B.ReadParameter_1.10:= AteqLeakageTester_B.Profinet_PLC_INPUTS[36].2;
    AteqLeakageTester_B.ReadParameter_1.11:= AteqLeakageTester_B.Profinet_PLC_INPUTS[36].3;
    AteqLeakageTester_B.ReadParameter_1.12:= AteqLeakageTester_B.Profinet_PLC_INPUTS[36].4;
    AteqLeakageTester_B.ReadParameter_1.13:= AteqLeakageTester_B.Profinet_PLC_INPUTS[36].5;
    AteqLeakageTester_B.ReadParameter_1.14:= AteqLeakageTester_B.Profinet_PLC_INPUTS[36].6;
    AteqLeakageTester_B.ReadParameter_1.15:= AteqLeakageTester_B.Profinet_PLC_INPUTS[36].7;

    AteqLeakageTester_B.ReadParameter_2.0:= AteqLeakageTester_B.Profinet_PLC_INPUTS[41].0;
    AteqLeakageTester_B.ReadParameter_2.1:= AteqLeakageTester_B.Profinet_PLC_INPUTS[41].1;
    AteqLeakageTester_B.ReadParameter_2.2:= AteqLeakageTester_B.Profinet_PLC_INPUTS[41].2;
    AteqLeakageTester_B.ReadParameter_2.3:= AteqLeakageTester_B.Profinet_PLC_INPUTS[41].3;
    AteqLeakageTester_B.ReadParameter_2.4:= AteqLeakageTester_B.Profinet_PLC_INPUTS[41].4;
    AteqLeakageTester_B.ReadParameter_2.5:= AteqLeakageTester_B.Profinet_PLC_INPUTS[41].5;
    AteqLeakageTester_B.ReadParameter_2.6:= AteqLeakageTester_B.Profinet_PLC_INPUTS[41].6;
    AteqLeakageTester_B.ReadParameter_2.7:= AteqLeakageTester_B.Profinet_PLC_INPUTS[41].7;
    AteqLeakageTester_B.ReadParameter_2.8:= AteqLeakageTester_B.Profinet_PLC_INPUTS[42].0;
    AteqLeakageTester_B.ReadParameter_2.9:= AteqLeakageTester_B.Profinet_PLC_INPUTS[42].1;
    AteqLeakageTester_B.ReadParameter_2.10:= AteqLeakageTester_B.Profinet_PLC_INPUTS[42].2;
    AteqLeakageTester_B.ReadParameter_2.11:= AteqLeakageTester_B.Profinet_PLC_INPUTS[42].3;
    AteqLeakageTester_B.ReadParameter_2.12:= AteqLeakageTester_B.Profinet_PLC_INPUTS[42].4;
    AteqLeakageTester_B.ReadParameter_2.13:= AteqLeakageTester_B.Profinet_PLC_INPUTS[42].5;
    AteqLeakageTester_B.ReadParameter_2.14:= AteqLeakageTester_B.Profinet_PLC_INPUTS[42].6;
    AteqLeakageTester_B.ReadParameter_2.15:= AteqLeakageTester_B.Profinet_PLC_INPUTS[42].7;

    AteqLeakageTester_B.ReadParameter_3.0:= AteqLeakageTester_B.Profinet_PLC_INPUTS[47].0;
    AteqLeakageTester_B.ReadParameter_3.1:= AteqLeakageTester_B.Profinet_PLC_INPUTS[47].1;
    AteqLeakageTester_B.ReadParameter_3.2:= AteqLeakageTester_B.Profinet_PLC_INPUTS[47].2;
    AteqLeakageTester_B.ReadParameter_3.3:= AteqLeakageTester_B.Profinet_PLC_INPUTS[47].3;
    AteqLeakageTester_B.ReadParameter_3.4:= AteqLeakageTester_B.Profinet_PLC_INPUTS[47].4;
    AteqLeakageTester_B.ReadParameter_3.5:= AteqLeakageTester_B.Profinet_PLC_INPUTS[47].5;
    AteqLeakageTester_B.ReadParameter_3.6:= AteqLeakageTester_B.Profinet_PLC_INPUTS[47].6;
    AteqLeakageTester_B.ReadParameter_3.7:= AteqLeakageTester_B.Profinet_PLC_INPUTS[47].7;
    AteqLeakageTester_B.ReadParameter_3.8:= AteqLeakageTester_B.Profinet_PLC_INPUTS[48].0;
    AteqLeakageTester_B.ReadParameter_3.9:= AteqLeakageTester_B.Profinet_PLC_INPUTS[48].1;
    AteqLeakageTester_B.ReadParameter_3.10:= AteqLeakageTester_B.Profinet_PLC_INPUTS[48].2;
    AteqLeakageTester_B.ReadParameter_3.11:= AteqLeakageTester_B.Profinet_PLC_INPUTS[48].3;
    AteqLeakageTester_B.ReadParameter_3.12:= AteqLeakageTester_B.Profinet_PLC_INPUTS[48].4;
    AteqLeakageTester_B.ReadParameter_3.13:= AteqLeakageTester_B.Profinet_PLC_INPUTS[48].5;
    AteqLeakageTester_B.ReadParameter_3.14:= AteqLeakageTester_B.Profinet_PLC_INPUTS[48].6;
    AteqLeakageTester_B.ReadParameter_3.15:= AteqLeakageTester_B.Profinet_PLC_INPUTS[48].7;

    AteqLeakageTester_B.ReadParameter_4.0:= AteqLeakageTester_B.Profinet_PLC_INPUTS[53].0;
    AteqLeakageTester_B.ReadParameter_4.1:= AteqLeakageTester_B.Profinet_PLC_INPUTS[53].1;
    AteqLeakageTester_B.ReadParameter_4.2:= AteqLeakageTester_B.Profinet_PLC_INPUTS[53].2;
    AteqLeakageTester_B.ReadParameter_4.3:= AteqLeakageTester_B.Profinet_PLC_INPUTS[53].3;
    AteqLeakageTester_B.ReadParameter_4.4:= AteqLeakageTester_B.Profinet_PLC_INPUTS[53].4;
    AteqLeakageTester_B.ReadParameter_4.5:= AteqLeakageTester_B.Profinet_PLC_INPUTS[53].5;
    AteqLeakageTester_B.ReadParameter_4.6:= AteqLeakageTester_B.Profinet_PLC_INPUTS[53].6;
    AteqLeakageTester_B.ReadParameter_4.7:= AteqLeakageTester_B.Profinet_PLC_INPUTS[53].7;
    AteqLeakageTester_B.ReadParameter_4.8:= AteqLeakageTester_B.Profinet_PLC_INPUTS[54].0;
    AteqLeakageTester_B.ReadParameter_4.9:= AteqLeakageTester_B.Profinet_PLC_INPUTS[54].1;
    AteqLeakageTester_B.ReadParameter_4.10:= AteqLeakageTester_B.Profinet_PLC_INPUTS[54].2;
    AteqLeakageTester_B.ReadParameter_4.11:= AteqLeakageTester_B.Profinet_PLC_INPUTS[54].3;
    AteqLeakageTester_B.ReadParameter_4.12:= AteqLeakageTester_B.Profinet_PLC_INPUTS[54].4;
    AteqLeakageTester_B.ReadParameter_4.13:= AteqLeakageTester_B.Profinet_PLC_INPUTS[54].5;
    AteqLeakageTester_B.ReadParameter_4.14:= AteqLeakageTester_B.Profinet_PLC_INPUTS[54].6;
    AteqLeakageTester_B.ReadParameter_4.15:= AteqLeakageTester_B.Profinet_PLC_INPUTS[54].7;

    AteqLeakageTester_B.ReadParameter_5.0:= AteqLeakageTester_B.Profinet_PLC_INPUTS[24].0;
    AteqLeakageTester_B.ReadParameter_5.1:= AteqLeakageTester_B.Profinet_PLC_INPUTS[24].1;
    AteqLeakageTester_B.ReadParameter_5.2:= AteqLeakageTester_B.Profinet_PLC_INPUTS[24].2;
    AteqLeakageTester_B.ReadParameter_5.3:= AteqLeakageTester_B.Profinet_PLC_INPUTS[24].3;
    AteqLeakageTester_B.ReadParameter_5.4:= AteqLeakageTester_B.Profinet_PLC_INPUTS[24].4;
    AteqLeakageTester_B.ReadParameter_5.5:= AteqLeakageTester_B.Profinet_PLC_INPUTS[24].5;
    AteqLeakageTester_B.ReadParameter_5.6:= AteqLeakageTester_B.Profinet_PLC_INPUTS[24].6;
    AteqLeakageTester_B.ReadParameter_5.7:= AteqLeakageTester_B.Profinet_PLC_INPUTS[24].7;
    AteqLeakageTester_B.ReadParameter_5.8:= AteqLeakageTester_B.Profinet_PLC_INPUTS[25].0;
    AteqLeakageTester_B.ReadParameter_5.9:= AteqLeakageTester_B.Profinet_PLC_INPUTS[25].1;
    AteqLeakageTester_B.ReadParameter_5.10:= AteqLeakageTester_B.Profinet_PLC_INPUTS[25].2;
    AteqLeakageTester_B.ReadParameter_5.11:= AteqLeakageTester_B.Profinet_PLC_INPUTS[25].3;
    AteqLeakageTester_B.ReadParameter_5.12:= AteqLeakageTester_B.Profinet_PLC_INPUTS[25].4;
    AteqLeakageTester_B.ReadParameter_5.13:= AteqLeakageTester_B.Profinet_PLC_INPUTS[25].5;
    AteqLeakageTester_B.ReadParameter_5.14:= AteqLeakageTester_B.Profinet_PLC_INPUTS[25].6;
    AteqLeakageTester_B.ReadParameter_5.15:= AteqLeakageTester_B.Profinet_PLC_INPUTS[25].7;
    AteqLeakageTester_B.ReadParameter_5.16:= AteqLeakageTester_B.Profinet_PLC_INPUTS[26].0;
    AteqLeakageTester_B.ReadParameter_5.17:= AteqLeakageTester_B.Profinet_PLC_INPUTS[26].1;
    AteqLeakageTester_B.ReadParameter_5.18:= AteqLeakageTester_B.Profinet_PLC_INPUTS[26].2;
    AteqLeakageTester_B.ReadParameter_5.19:= AteqLeakageTester_B.Profinet_PLC_INPUTS[26].3;
    AteqLeakageTester_B.ReadParameter_5.20:= AteqLeakageTester_B.Profinet_PLC_INPUTS[26].4;
    AteqLeakageTester_B.ReadParameter_5.21:= AteqLeakageTester_B.Profinet_PLC_INPUTS[26].5;
    AteqLeakageTester_B.ReadParameter_5.22:= AteqLeakageTester_B.Profinet_PLC_INPUTS[26].6;
    AteqLeakageTester_B.ReadParameter_5.23:= AteqLeakageTester_B.Profinet_PLC_INPUTS[26].7;
    AteqLeakageTester_B.ReadParameter_5.24:= AteqLeakageTester_B.Profinet_PLC_INPUTS[27].0;
    AteqLeakageTester_B.ReadParameter_5.25:= AteqLeakageTester_B.Profinet_PLC_INPUTS[27].1;
    AteqLeakageTester_B.ReadParameter_5.26:= AteqLeakageTester_B.Profinet_PLC_INPUTS[27].2;
    AteqLeakageTester_B.ReadParameter_5.27:= AteqLeakageTester_B.Profinet_PLC_INPUTS[27].3;
    AteqLeakageTester_B.ReadParameter_5.28:= AteqLeakageTester_B.Profinet_PLC_INPUTS[27].4;
    AteqLeakageTester_B.ReadParameter_5.29:= AteqLeakageTester_B.Profinet_PLC_INPUTS[27].5;
    AteqLeakageTester_B.ReadParameter_5.30:= AteqLeakageTester_B.Profinet_PLC_INPUTS[27].6;
    AteqLeakageTester_B.ReadParameter_5.31:= AteqLeakageTester_B.Profinet_PLC_INPUTS[27].7;

	//Vystupy z PLC do Testera//
	AteqLeakageTester_B.Profinet_PLC_OUTPUTS[1].0:= AteqLeakageTester_B.RESET_Vysledkov;
	AteqLeakageTester_B.Profinet_PLC_OUTPUTS[1].1:= AteqLeakageTester_B.START_Testovania;
	AteqLeakageTester_B.Profinet_PLC_OUTPUTS[1].3:= AteqLeakageTester_B.ZMEN_Program;
	AteqLeakageTester_B.Profinet_PLC_OUTPUTS[1].5:= AteqLeakageTester_B.CitajParametreTestera;

	AteqLeakageTester_B.Profinet_PLC_OUTPUTS[7].0:= AteqLeakageTester_B.CisloZadanehoProgramu.0;
	AteqLeakageTester_B.Profinet_PLC_OUTPUTS[7].1:= AteqLeakageTester_B.CisloZadanehoProgramu.1;
	AteqLeakageTester_B.Profinet_PLC_OUTPUTS[7].2:= AteqLeakageTester_B.CisloZadanehoProgramu.2;
	AteqLeakageTester_B.Profinet_PLC_OUTPUTS[7].3:= AteqLeakageTester_B.CisloZadanehoProgramu.3;
	AteqLeakageTester_B.Profinet_PLC_OUTPUTS[7].4:= AteqLeakageTester_B.CisloZadanehoProgramu.4;
	AteqLeakageTester_B.Profinet_PLC_OUTPUTS[7].5:= AteqLeakageTester_B.CisloZadanehoProgramu.5;
	AteqLeakageTester_B.Profinet_PLC_OUTPUTS[7].6:= AteqLeakageTester_B.CisloZadanehoProgramu.6;
	AteqLeakageTester_B.Profinet_PLC_OUTPUTS[7].7:= AteqLeakageTester_B.CisloZadanehoProgramu.7;

	AteqLeakageTester_B.Profinet_PLC_OUTPUTS[8].0:= AteqLeakageTester_B.CisloZadanehoProgramu.8;
	AteqLeakageTester_B.Profinet_PLC_OUTPUTS[8].1:= AteqLeakageTester_B.CisloZadanehoProgramu.9;
	AteqLeakageTester_B.Profinet_PLC_OUTPUTS[8].2:= AteqLeakageTester_B.CisloZadanehoProgramu.10;
	AteqLeakageTester_B.Profinet_PLC_OUTPUTS[8].3:= AteqLeakageTester_B.CisloZadanehoProgramu.11;
	AteqLeakageTester_B.Profinet_PLC_OUTPUTS[8].4:= AteqLeakageTester_B.CisloZadanehoProgramu.12;
	AteqLeakageTester_B.Profinet_PLC_OUTPUTS[8].5:= AteqLeakageTester_B.CisloZadanehoProgramu.13;
	AteqLeakageTester_B.Profinet_PLC_OUTPUTS[8].6:= AteqLeakageTester_B.CisloZadanehoProgramu.14;
	AteqLeakageTester_B.Profinet_PLC_OUTPUTS[8].7:= AteqLeakageTester_B.CisloZadanehoProgramu.15;

    AteqLeakageTester_B.PocetCitanychParametrov:= 4;
    AteqLeakageTester_B.IdentifikaciaParametra_1:= 1;
    AteqLeakageTester_B.IdentifikaciaParametra_2:= 2;
    AteqLeakageTester_B.IdentifikaciaParametra_3:= 66;
    AteqLeakageTester_B.IdentifikaciaParametra_4:= 60;

    //Vyčítané parametre//
    CasPneniaREAL:= UINT_TO_REAL(AteqLeakageTester_B.ReadParameter_1);
    AteqLeakageTester_B.CasPnenia:= CasPneniaREAL/1000;
    CasStabilizacieREAL:= UINT_TO_REAL(AteqLeakageTester_B.ReadParameter_2);
    AteqLeakageTester_B.CasStabilizacie:= CasStabilizacieREAL/1000;
    TlakPlneniaREAL:= UINT_TO_REAL(AteqLeakageTester_B.ReadParameter_3);
    AteqLeakageTester_B.TlakPlnenia:= TlakPlneniaREAL/1000;
    ToleranciaREAL:= UINT_TO_REAL(AteqLeakageTester_B.ReadParameter_4);
    AteqLeakageTester_B.Tolerancia:= ToleranciaREAL/1000;
    TlakUnikuREAL:= DINT_TO_REAL(AteqLeakageTester_B.ReadParameter_5);
    AteqLeakageTester_B.TlakUniku:= ((TlakUnikuREAL/1000)*6)/1536;

END_ACTION
```

### Program Logical/Program/Pracovisko_3/P34_OvladanieVizu (IEC)
